// TwinCAT 3 PLC project cryo
// Title: ESO LDC Cryo Library
// Company: ESO
// ProjectVersion: 0.0.0.10
// ProgramVersion: 3.1.4022.4
// libraries:
//   ESO LDC Comm Tcp Library, * (ESO)
//   Tc2_SerialCom, * (Beckhoff Automation GmbH)
//   Tc2_Standard, * (Beckhoff Automation GmbH)
//   Tc2_System, * (Beckhoff Automation GmbH)
//   Tc2_Utilities, * (Beckhoff Automation GmbH)
//   Tc3_Module, * (Beckhoff Automation GmbH)
//   VisuDialogs, * (System)
//   ESO LDC Comm Common Library,0.2.0.2,ESO
//   ESO LDC Comm Serial Library,0.2.0.2,ESO
//   VisuSymbols,3.5.10.0,System
// project tree:
//   / ClassDiagram.TcCD (not stored), ClassDiagram_All.TcCD (not stored), ClassDiagram_Sensors.TcCD (not stored), GlobalTextList.TcGTLO, ImagePool.TcIPO (not stored), PlcTask.TcTTO, Visualization Manager.TcVMO (not stored)
//   DUTs/Enumerations/Actuators/ E_CRYO_BIN_ACT_CMD.TcDUT, E_CRYO_BIN_ACT_FEEDBACK.TcDUT, E_CRYO_BIN_ACT_FEEDBACK_STATE.TcDUT, E_CRYO_BIN_ACT_STATE.TcDUT, E_CRYO_BIN_CTRL_ACTION.TcDUT, E_CRYO_BIN_CTRL_STATE.TcDUT, E_CRYO_CTRL_CMD.TcDUT, E_CRYO_CTRL_STATE.TcDUT, E_CRYO_GEN_CTRL_EVENT.TcDUT
//   DUTs/Enumerations/Coolers/ E_CRYO_CPA_ALARM.TcDUT, E_CRYO_CPA_CMDS.TcDUT, E_CRYO_CPA_DIAG_IDX.TcDUT, E_CRYO_CRYOTELGT_CMD.TcDUT, E_CRYO_CRYOTELGT_STATE.TcDUT
//   DUTs/Enumerations/Misc/ E_CRYO_ALARM_IDX.TcDUT, E_CRYO_ALARM_LEVEL.TcDUT, E_CRYO_THLD_MODE.TcDUT, E_CRYO_VOTE.TcDUT
//   DUTs/Enumerations/Pumps/ E_CRYO_PUMP_STATE.TcDUT, E_ECODRY_VERSION.TcDUT
//   DUTs/Enumerations/Sensors/ E_CRYO_SBG232_SENSOR_TYPE.TcDUT, E_CRYO_SENSOR_TYPE_PRESS.TcDUT, E_CRYO_SENSOR_TYPE_TEMP.TcDUT, E_CRYO_SIM_SENS_CMD.TcDUT
//   DUTs/Enumerations/Subsystems/Evacuation/ E_CRYO_EVAC_PRESSURES_50000.TcDUT, E_CRYO_EVAC_STATE.TcDUT, E_CRYO_EVAC_STATE_50000.TcDUT, E_CRYO_EVAC_SYS_STATE.TcDUT, E_CRYO_EVAC_VALVES_50000.TcDUT
//   DUTs/Structures/Actuators/ T_CRYO_BIN_ACT_STATUS.TcDUT, T_CRYO_BIN_CTRL_STATUS.TcDUT, T_CRYO_GEN_CTRL_STATUS_BASE.TcDUT
//   DUTs/Structures/Coolers/ T_CRYO_CPA_ACTIVE_LIMITS.TcDUT, T_CRYO_CPA_CFG.TcDUT, T_CRYO_CPA_CTRL.TcDUT, T_CRYO_CPA_DIAG_CFG.TcDUT, T_CRYO_CPA_INFO.TcDUT, T_CRYO_CPA_STAT.TcDUT, T_CRYO_CRYOTELGT_CFG.TcDUT, T_CRYO_CRYOTELGT_CMD.TcDUT, T_CRYO_CRYOTELGT_CTRL.TcDUT, T_CRYO_CRYOTELGT_STAT.TcDUT
//   DUTs/Structures/Misc/ T_CRYO_VOTE_LIST.TcDUT
//   DUTs/Structures/Pumps/ T_CRYO_PUMP_ATM2303M_CFG.TcDUT, T_CRYO_PUMP_ATM2303M_STAT.TcDUT, T_CRYO_PUMP_BASE_CFG.TcDUT, T_CRYO_PUMP_BASE_CTRL.TcDUT, T_CRYO_PUMP_BASE_STAT.TcDUT, T_CRYO_PUMP_CMD.TcDUT, T_CRYO_PUMP_HIPACE30_CFG.TcDUT, T_CRYO_PUMP_HIPACE30_STAT.TcDUT, T_CRYO_PUMP_MODBUS_CFG.TcDUT, T_CRYO_PUMP_MODBUS_CTRL.TcDUT, T_CRYO_PUMP_MODBUS_STAT.TcDUT, T_CRYO_PUMP_MVP030_CFG.TcDUT, T_CRYO_PUMP_MVP030_STAT.TcDUT, T_CRYO_PUMP_SERIAL_CFG.TcDUT
//   DUTs/Structures/Sensors/ T_CRYO_IOLINK_SENSOR_STATUS.TcDUT, T_CRYO_PRESSURE_STATUS.TcDUT, T_CRYO_PRESSURE_VOTE_STATUS.TcDUT, T_CRYO_PT100_OHM2C_REC.TcDUT, T_CRYO_SBG232_STAT.TcDUT, T_CRYO_SENSOR_STATUS.TcDUT, T_CRYO_SENSOR_STATUS_PRESS.TcDUT, T_CRYO_SENSOR_STATUS_TEMP.TcDUT, T_CRYO_TEMPERATURE_STATUS.TcDUT
//   DUTs/Structures/Subsystems/Evacuation/ T_CRYO_EVACUATION_SYSTEM_STATUS.TcDUT, T_CRYO_EVAC_CFG.TcDUT, T_CRYO_EVAC_CFG_50000.TcDUT, T_CRYO_EVAC_CTRL.TcDUT, T_CRYO_EVAC_CTRL_50000.TcDUT, T_CRYO_EVAC_STAT.TcDUT, T_CRYO_EVAC_STAT_50000.TcDUT, T_CRYO_EVAC_SYS_INPUT.TcDUT
//   DUTs/Structures/System/ T_CRYO_CFG.TcDUT, T_CRYO_CTRL.TcDUT, T_CRYO_LOG.TcDUT, T_CRYO_STAT.TcDUT
//   POUs/Actuators/ FB_CRYO_ACTUATOR_CMD.TcPOU, FB_CRYO_CMD_OVERRIDE.TcPOU, FB_CRYO_BIN_ACT.TcPOU, FB_CRYO_BIN_CTRL.TcPOU, FB_CRYO_GEN_CTRL_BASE.TcPOU, FB_CRYO_CCC_CTRL.TcPOU, FB_CRYO_HEATER_CTRL.TcPOU, FB_CRYO_LN2_CTRL.TcPOU, FB_CRYO_VALVE_CTRL.TcPOU
//   POUs/Comm/ FB_MODBUS_COMM_CPA.TcPOU
//   POUs/Coolers/ FB_CRYO_CPA.TcPOU, FB_CRYO_CRYOTELGT.TcPOU, FB_RS_COMM_CRYOTELGT.TcPOU, FB_SIM_RS_COMM_CRYOTELGT.TcPOU
//   POUs/ MAIN.TcPOU
//   POUs/Pumps/ FB_CRYO_PUMP_ATH2303M.TcPOU, FB_CRYO_PUMP_BASE.TcPOU, FB_CRYO_PUMP_ECODRY.TcPOU, FB_CRYO_PUMP_HIPACE30.TcPOU, FB_CRYO_PUMP_MODBUS.TcPOU, FB_CRYO_PUMP_MVP030.TcPOU, FB_CRYO_PUMP_SERIAL.TcPOU
//   POUs/Sensors/ FB_CRYO_PRESSURE.TcPOU, FB_CRYO_PRESSURE_VOTE.TcPOU, FB_CRYO_SBG232.TcPOU, FB_CRYO_SENSOR_BASE.TcPOU, FB_CRYO_SENSOR_PRESSURE.TcPOU, FB_CRYO_SENSOR_TEMPERATURE.TcPOU, FB_CRYO_TEMPERATURE.TcPOU
//   POUs/Simulation/ FB_CRYO_SIM_CTRL.TcPOU, FB_CRYO_SIM_SBG232.TcPOU, FB_CRYO_SIM_TEMPERATURE.TcPOU, FB_CRYO_SIM_PRESSURE.TcPOU, FB_CRYO_SIM_SINE.TcPOU, FB_SIM_MODBUS_COMM_CPA.TcPOU
//   POUs/Subsystems/Evacuation/ FB_CRYO_EVACUATION_SYSTEM.TcPOU, FB_CRYO_EVAC_BASE.TcPOU, FB_CRYO_EVAC_BASE_50000.TcPOU
//   POUs/Subsystems/Examples/Evacuation/ FB_CRYO_EVAC_ECODRY_ATH2303M.TcPOU, FB_CRYO_EVAC_MICADO.TcPOU, FB_CRYO_EVAC_PDS.TcPOU, FB_SIM_MICADO_PUMPS.TcPOU, FB_SIM_MICADO_VALVES.TcPOU
//   POUs/Subsystems/Examples/LN2_Precooling/ FB_CRYO_LN2_PRECOOL.TcPOU, FB_SIM_LN2_PRECOOL.TcPOU
//   POUs/System/ FB_CRYO_CTRL.TcPOU
//   POUs/Utilities/ FB_CRYO_THLD_BASE.TcPOU
//   VISUs/GUIs/ GUI_ATH2303M_EVAC_LAB.TcVIS, GUI_CMD_OVERRIDE.TcVIS, GUI_CPA.TcVIS, GUI_CRYO.TcVIS, GUI_CRYOTELGT.TcVIS, GUI_ECODRY_V01_EVAC_LAB.TcVIS, GUI_EVAC_LAB.TcVIS, GUI_EVAC_MICADO.TcVIS, GUI_EVAC_PDS.TcVIS, GUI_HIPACE_30_EVAC_PDS.TcVIS, GUI_IRATEC.TcVIS, GUI_MICADO_Valves.TcVIS, GUI_MVP030_EVAC_PDS.TcVIS, GUI_P2_OVERRIDE.TcVIS, GUI_Pressures.TcVIS, GUI_PVV1_CMD.TcVIS, GUI_SBG232.TcVIS, GUI_SBG232_SIM.TcVIS, GUI_T2_OVERRIDE.TcVIS
//   VISUs/Templates/ GUI_TEMPLATE_ACTUATOR_CMD.TcVIS, GUI_TEMPLATE_ACTUATOR_ENG.TcVIS, GUI_TEMPLATE_SENSOR_SIM_OVERRIDE.TcVIS, GUI_TEMPLATE_ATH2303M.TcVIS, GUI_TEMPLATE_CMD_OVERRIDE.TcVIS, GUI_TEMPLATE_CRYOTELGT.TcVIS, GUI_TEMPLATE_CRYO_CPA.TcVIS, GUI_TEMPLATE_CRYO_EVAC_BASE.TcVIS, GUI_TEMPLATE_ECODRY_V01.TcVIS, GUI_TEMPLATE_HIPACE_30.TcVIS, GUI_TEMPLATE_MVP030.TcVIS, GUI_TEMPLATE_SBG232.TcVIS, GUI_TEMPLATE_TEMP_OVERRIDE.TcVIS, GUI_TEMPLATE_PRESS_OVERRIDE.TcVIS
// real-time tasks:
//   TASK PlcTask: cycle T#1ms, priority 20, ADS port 350
//   TASK VISU_TASK: cycle T#200000us, priority 30, ADS port 351
// motion (NC):
//   TASK NC-Task 1 SAF: cycle T#2ms, priority 4, ADS port 501
//   TASK NC-Task 1 SVB: cycle T#10ms, priority 8, ADS port 511
// I/O:
//   DEVICE Device 1 (EtherCAT) (disabled), AmsNetId 134.171.34.120.2.1
//     Term 1 (EK1200) [EK1200-5000 EtherCAT Power supply (2A E-Bus)]
//       Term 2 (EL2008) [EL2008 8Ch. Dig. Output 24V, 0.5A]
//       Term 3 (EL3162) [EL3162 2Ch. Ana. Input 0-10V]
//       Term 4 (EL1004) [EL1004 4Ch. Dig. Input 24V, 3ms]
//       Term 5 (EL1004) [EL1004 4Ch. Dig. Input 24V, 3ms]
//       Term 6 (EL2622) [EL2622 2Ch. Relay Output, NO (230V AC / 30V DC)]
//       Term 7 (EL6022) [EL6022 Interface 2Ch. (RS422/485)]
//       Term 8 (EL6002) [EL6002 Interface 2Ch. (RS232)]
//       Term 9 (EL9011) [EL9011 End Terminal]
//   DEVICE Device 5 (EtherCAT) (disabled), AmsNetId 134.171.34.120.6.1
//     Term 10 (EK1100) [EK1100 EtherCAT Coupler (2A E-Bus)]
//       Term 11 (EL6224) [EL6224 (IO Link Master)]
//       Term 12 (EL1808) [EL1808 8Ch. Dig. Input 24V, 3ms]
//       Term 13 (EL1808) [EL1808 8Ch. Dig. Input 24V, 3ms]
//       Term 14 (EL2808) [EL2808 8Ch. Dig. Output 24V, 0.5A]
//       Term 15 (EL2652) [EL2652 2Ch. Relay Output, CO (230V AC / 30V DC)]
//       Term 16 (EL2652) [EL2652 2Ch. Relay Output, CO (230V AC / 30V DC)]
//       Term 17 (EL6022) [EL6022 Interface 2Ch. (RS422/485)]
//       Term 18 (EL6022) [EL6022 Interface 2Ch. (RS422/485)]
//       Term 10 (EL9011) [EL9011 End Terminal]
// variable links:
//   cryo/cryo Instance <-> cryo/cryo Instance
//     PlcTask Inputs/MAIN.evac_micado.GBV.Actuator.i_bOFF <-> PlcTask Outputs/MAIN.mic_valves.q_bOFF_GBV
//     PlcTask Inputs/MAIN.evac_micado.GBV.Actuator.i_bON <-> PlcTask Outputs/MAIN.mic_valves.q_bON_GBV
//     PlcTask Inputs/MAIN.evac_micado.GBV.Actuator.i_nCouplerState <-> PlcTask Outputs/MAIN.q_nCouplerState
//     PlcTask Inputs/MAIN.evac_micado.PVV{1..4}.Actuator.i_bOFF <-> PlcTask Outputs/MAIN.mic_valves.q_bOFF_PVV{1..4}  (4 links)
//     PlcTask Inputs/MAIN.evac_micado.PVV{1..4}.Actuator.i_bON <-> PlcTask Outputs/MAIN.mic_valves.q_bON_PVV{1..4}  (4 links)
//     PlcTask Inputs/MAIN.evac_micado.PVV{1..4}.Actuator.i_nCouplerState <-> PlcTask Outputs/MAIN.q_nCouplerState  (4 links)
//     PlcTask Inputs/MAIN.evac_micado.rp.i_bRunning <-> PlcTask Outputs/MAIN.mic_pumps.q_PVP_Running
//     PlcTask Inputs/MAIN.evac_micado.sensor_VAG1.i_nStatus <-> PlcTask Outputs/MAIN.pSim.q_nStatus
//     PlcTask Inputs/MAIN.evac_micado.sensor_VAG2.i_nStatus <-> PlcTask Outputs/MAIN.pSim.q_nStatus
//     PlcTask Inputs/MAIN.evac_micado.sensor_VAG3.i_nStatus <-> PlcTask Outputs/MAIN.pSim.q_nStatus
//     PlcTask Inputs/MAIN.evac_micado.sensor_VAG1.i_nValue <-> PlcTask Outputs/MAIN.q_nVAG1
//     PlcTask Inputs/MAIN.evac_micado.sensor_VAG2.i_nValue <-> PlcTask Outputs/MAIN.q_nVAG2
//     PlcTask Inputs/MAIN.evac_micado.sensor_VAG3.i_nValue <-> PlcTask Outputs/MAIN.q_nVAG3
//     PlcTask Inputs/MAIN.evac_micado.tp.i_bReady <-> PlcTask Outputs/MAIN.mic_pumps.q_TMP_Ready
//     PlcTask Inputs/MAIN.evac_micado.tp.i_bSpeed100 <-> PlcTask Outputs/MAIN.mic_pumps.q_TMP_Speed100
//     PlcTask Inputs/MAIN.ln2_ctrl.valve.Actuator.i_bON <-> PlcTask Outputs/MAIN.ln2_ctrl.valve.Actuator.q_bCtrl
//     PlcTask Inputs/MAIN.ln2_ctrl.valve.Actuator.i_nCouplerState <-> PlcTask Outputs/MAIN.Cryo_Ctrl.q_nStateDummy
//     PlcTask Inputs/MAIN.mic_valves.i_bON_GBV <-> PlcTask Outputs/MAIN.evac_micado.GBV.Actuator.q_bCtrl
//     PlcTask Inputs/MAIN.mic_valves.i_bON_PVV{1..4} <-> PlcTask Outputs/MAIN.evac_micado.PVV{1..4}.Actuator.q_bCtrl  (4 links)
//     PlcTask Inputs/MAIN.sbg232_sim.i_ArrPortProcessData <-> PlcTask Outputs/MAIN.SIM_sbg232.q_ArrPortProcessData
//     PlcTask Inputs/MAIN.sbg232_sim.i_nCouplerState <-> PlcTask Outputs/MAIN.SIM_sbg232.q_nCouplerState
//     PlcTask Inputs/MAIN.sbg232_sim.i_nDeviceStateInputCh <-> PlcTask Outputs/MAIN.SIM_sbg232.q_nDeviceStateInputCh
//     PlcTask Inputs/MAIN.sensor_VAGF1.i_nStatus <-> PlcTask Outputs/MAIN.pSim.q_nStatus
//     PlcTask Inputs/MAIN.sensor_VAGF2.i_nStatus <-> PlcTask Outputs/MAIN.pSim.q_nStatus
//     PlcTask Inputs/MAIN.sensor_VAGF1.i_nValue <-> PlcTask Outputs/MAIN.q_nVAGF1
//     PlcTask Inputs/MAIN.sensor_VAGF2.i_nValue <-> PlcTask Outputs/MAIN.q_nVAGF2
//     PlcTask Inputs/MAIN.sensor_VAGG1.i_nStatus <-> PlcTask Outputs/MAIN.pSim.q_nStatus
//     PlcTask Inputs/MAIN.sensor_VAGG2.i_nStatus <-> PlcTask Outputs/MAIN.pSim.q_nStatus
//     PlcTask Inputs/MAIN.sensor_VAGG1.i_nValue <-> PlcTask Outputs/MAIN.q_nVAGG1
//     PlcTask Inputs/MAIN.sensor_VAGG2.i_nValue <-> PlcTask Outputs/MAIN.q_nVAGG2

CONFIGURATION cryo
    RESOURCE PLC ON TwinCAT3
        TASK PlcTask(INTERVAL := T#1ms, PRIORITY := 20);
        PROGRAM MAIN WITH PlcTask : MAIN;
    END_RESOURCE
END_CONFIGURATION

// ---- DUTs/Enumerations/Actuators/E_CRYO_BIN_ACT_CMD.TcDUT
{attribute 'qualified_only'}
{attribute 'strict'}
TYPE E_CRYO_BIN_ACT_CMD :
(
	NONE	:= 0,
	OFF 	:= 1,
	ON		:= 2
);
END_TYPE

// ---- DUTs/Enumerations/Actuators/E_CRYO_BIN_ACT_FEEDBACK.TcDUT
{attribute 'qualified_only'}
{attribute 'strict'}
TYPE E_CRYO_BIN_ACT_FEEDBACK :
(
	ON_AND_OFF	:= 0,	// There are two separate signals: ON (i_bON) and OFF (i_bOFF)
	ON_ONLY 	:= 1	// Feedback exists only for ON signal
);
END_TYPE

// ---- DUTs/Enumerations/Actuators/E_CRYO_BIN_ACT_FEEDBACK_STATE.TcDUT
{attribute 'qualified_only'}
{attribute 'strict'}
TYPE E_CRYO_BIN_ACT_FEEDBACK_STATE :
(
	OFF		:= 0,
	ON	 	:= 1,
	ERROR	:= 2
);
END_TYPE

// ---- DUTs/Enumerations/Actuators/E_CRYO_BIN_ACT_STATE.TcDUT
{attribute 'qualified_only'}
{attribute 'strict'}
TYPE E_CRYO_BIN_ACT_STATE :
(
	NONE := 0,
	OFF,
	SWITCHING_ON,
	ON,
	SWITCHING_OFF,
	ERROR
);
END_TYPE

// ---- DUTs/Enumerations/Actuators/E_CRYO_BIN_CTRL_ACTION.TcDUT
TYPE E_CRYO_BIN_CTRL_ACTION :
(
	NONE := 0,
	OFF,
	ON
);
END_TYPE

// ---- DUTs/Enumerations/Actuators/E_CRYO_BIN_CTRL_STATE.TcDUT
{attribute 'qualified_only'}
{attribute 'strict'}
TYPE E_CRYO_BIN_CTRL_STATE :
(
	NONE := 0,
	OFF,					// Controller OFF, Actuator OFF
	ACTIVE_SWITCHING_ON,	// Activating Controller
	ACTIVE_OFF,				// Controller active, Actuator OFF
	ACTIVE_ON,				// Controller active, Actuator ON
	ACTIVE_SWITCHING_OFF,	// Switching Actuator OFF and going OFF with Controller
	ERROR					// Actuator failure
);
END_TYPE

// ---- DUTs/Enumerations/Actuators/E_CRYO_CTRL_CMD.TcDUT
{attribute 'qualified_only'}
{attribute 'strict'}
TYPE E_CRYO_CTRL_CMD :
(
	NONE	:= 0,
	PRECOOL,
	COOL,
	WARM_UP,
	REPRESSURIZE
);
END_TYPE

// ---- DUTs/Enumerations/Actuators/E_CRYO_CTRL_STATE.TcDUT
{attribute 'qualified_only'}
{attribute 'strict'}
TYPE E_CRYO_CTRL_STATE :
(
	NONE 			:= 0,
	WARM_PRESS,				// Warm & Pressurized
	WARM_VACUUM,			// Warm & Vacuum
	PRE_COOLING,			// Pre_cooling
	PRE_COOLED,				// Pre_cooled
	COOLING_DOWN,			// Cooling down
	COLD,					// Cold, i.e. fully operational
	WARMING_UP,				// Warming up
	REPRESSURIZING,			// Re-pressurizing			
	ERROR					// Controller failure
);
END_TYPE

// ---- DUTs/Enumerations/Actuators/E_CRYO_GEN_CTRL_EVENT.TcDUT
{attribute 'qualified_only'}
{attribute 'strict'}
TYPE E_CRYO_GEN_CTRL_EVENT :
(
	NONE := 0,
	ENABLE,
	DISABLE,
	OFF,
	IS_OFF,
	ON,
	IS_ON,
	ERROR
);
END_TYPE

// ---- DUTs/Enumerations/Coolers/E_CRYO_CPA_ALARM.TcDUT
{attribute 'qualified_only'}
{attribute 'strict'}
TYPE E_CRYO_CPA_ALARM :
(
	NONE := 0,
	LOW,
	HIGH
);
END_TYPE

// ---- DUTs/Enumerations/Coolers/E_CRYO_CPA_CMDS.TcDUT
{attribute 'qualified_only'}
{attribute 'strict'}
TYPE E_CRYO_CPA_CMDS :
(
	NONE	:= 0,
	START	:= 21,
	STOP
);
END_TYPE

// ---- DUTs/Enumerations/Coolers/E_CRYO_CPA_DIAG_IDX.TcDUT
{attribute 'qualified_only'}
{attribute 'strict'}
TYPE E_CRYO_CPA_DIAG_IDX :
(
	WATER_IN	:= 0,
	WATER_OUT,
	OIL_TEMP,
	HELIUM_TEMP,
	HELIUM_LOW_PRESS_OP,
	HELIUM_HIGH_PRESS_OP,
	HELIUM_DELTA_PRESS,
	HELIUM_STATIC_LOW_PRESS,
	HELIUM_STATIC_HIGH_PRESS
);
END_TYPE

// ---- DUTs/Enumerations/Coolers/E_CRYO_CRYOTELGT_CMD.TcDUT
{attribute 'qualified_only'}
{attribute 'strict'}
TYPE E_CRYO_CRYOTELGT_CMD :
(
	NONE := 0,
	OFF,
	ON,
	SET_POWER
);
END_TYPE

// ---- DUTs/Enumerations/Coolers/E_CRYO_CRYOTELGT_STATE.TcDUT
{attribute 'qualified_only'}
{attribute 'strict'}
TYPE E_CRYO_CRYOTELGT_STATE :
(
	OFF := 0,
	STARTING,
	ON,
	STOPPING,
	ERROR
);
END_TYPE

// ---- DUTs/Enumerations/Misc/E_CRYO_ALARM_IDX.TcDUT
{attribute 'qualified_only'}
{attribute 'strict'}
TYPE E_CRYO_ALARM_IDX :
(
	ALARM_LOW 		:= 1,
	WARNING_LOW		:= 2,
	WARNING_HIGH	:= 3,
	ALARM_HIGH		:= 4
);
END_TYPE

// ---- DUTs/Enumerations/Misc/E_CRYO_ALARM_LEVEL.TcDUT
{attribute 'qualified_only'}
{attribute 'strict'}
TYPE E_CRYO_ALARM_LEVEL :
(
	ALARM_LOW 		:= -2,
	WARNING_LOW		:= -1,
	NORMAL			:= 0,
	WARNING_HIGH	:= 1,
	ALARM_HIGH		:= 2
);
END_TYPE

// ---- DUTs/Enumerations/Misc/E_CRYO_THLD_MODE.TcDUT
{attribute 'qualified_only'}
{attribute 'strict'}
TYPE E_CRYO_THLD_MODE :
(
	FIXED := 0,		// Thresholds as set with input parameters
	ACTIVE,			// Thresholds are calculated based on input parameter(s)
	LAST_ACTIVE		// Thresholds are kept at last ACTIVE levels 
);
END_TYPE

// ---- DUTs/Enumerations/Misc/E_CRYO_VOTE.TcDUT
{attribute 'qualified_only'}
{attribute 'strict'}
TYPE E_CRYO_VOTE :
(
	V_AVE	:= 0,
	V_MIN,
	V_MAX,
	V_1oo2,
	V_2oo3,
	V_3oo5
);
END_TYPE

// ---- DUTs/Enumerations/Pumps/E_CRYO_PUMP_STATE.TcDUT
{attribute 'qualified_only'}
{attribute 'strict'}
TYPE E_CRYO_PUMP_STATE :
(
	OFF := 0,
	STARTING,
	ON,
	STOPPING,
	ERROR
);
END_TYPE

// ---- DUTs/Enumerations/Pumps/E_ECODRY_VERSION.TcDUT
{attribute 'qualified_only'}
{attribute 'strict'}
TYPE E_ECODRY_VERSION :
(
	V01 := 0,
	V21_22
);
END_TYPE

// ---- DUTs/Enumerations/Sensors/E_CRYO_SBG232_SENSOR_TYPE.TcDUT
{attribute 'qualified_only'}
{attribute 'strict'}
TYPE E_CRYO_SBG232_SENSOR_TYPE :
(
	NONE := 0,
	FLOW,
	TEMP
);
END_TYPE

// ---- DUTs/Enumerations/Sensors/E_CRYO_SENSOR_TYPE_PRESS.TcDUT
{attribute 'qualified_only'}
{attribute 'strict'}
TYPE E_CRYO_SENSOR_TYPE_PRESS :
(
	NONE 		:= 0,
	PKR_250		:= 1,	// Pfeiffer PKR250 & PKR251 have the same formula
	CMR_361		:= 2,	// Pfeiffer CMR361
	WRG_D_NW25	:= 3,	// Edwards WRG-D-NW25
	PKR_360		:= 4	// Pfeiffer PKR360
);
END_TYPE

// ---- DUTs/Enumerations/Sensors/E_CRYO_SENSOR_TYPE_TEMP.TcDUT
{attribute 'qualified_only'}
{attribute 'strict'}
TYPE E_CRYO_SENSOR_TYPE_TEMP :
(
	NONE 	:= 0,
	PT100	:= 1
);
END_TYPE

// ---- DUTs/Enumerations/Sensors/E_CRYO_SIM_SENS_CMD.TcDUT
{attribute 'qualified_only'}
{attribute 'strict'}
TYPE E_CRYO_SIM_SENS_CMD :
(
	NONE	:= 0,
	SET 	:= 1,	// Set value
	RAMP	:= 2,	// Ramp value
	SINE	:= 3	// Vary value as SINE signal
);
END_TYPE

// ---- DUTs/Enumerations/Subsystems/Evacuation/E_CRYO_EVAC_PRESSURES_50000.TcDUT
{attribute 'qualified_only'}
{attribute 'strict'}
TYPE E_CRYO_EVAC_PRESSURES_50000 :
(
	NONE := 0,
	VAG1,		
	VAG2,		
	VAG3,		
	VAGF,		
	VAGG		
);
END_TYPE

// ---- DUTs/Enumerations/Subsystems/Evacuation/E_CRYO_EVAC_STATE.TcDUT
{attribute 'qualified_only'}
{attribute 'strict'}
TYPE E_CRYO_EVAC_STATE :
(
	NONE := 0,				// Undefined state.
	OFF,					// Everything is OFF.
	START_R_PUMP,			// Starting Roughing Pump.
	WAIT_PREVAC,			// Waiting for the prevaccum pressure to be reached.
	OPEN_INSULATION_VALVE,	// Opening Insulation Valve.
	START_T_PUMP,			// Starting Turbo-Molecular Pump.
	WAIT_CRYO_VAC,			// Waiting for the cryo pressure to drop below threshold.
	EVACUATING,				// System is running. Evacuation in progress.
	CLOSE_INSULATION_VALVE,	// Closing Insulation Valve.
	DELAY_STOPPING,			// Delay after closing Insulation valve before stopping pumps.
	STOP_T_PUMP,			// Stopping Turbo-Molecular Pump.
	STOP_R_PUMP,			// Stopping Roughing Pump.
	WAIT_T_PUMP_STOP		// Waiting for the Turbo-Molecular Pump to stop.
);
END_TYPE

// ---- DUTs/Enumerations/Subsystems/Evacuation/E_CRYO_EVAC_STATE_50000.TcDUT
{attribute 'qualified_only'}
{attribute 'strict'}
TYPE E_CRYO_EVAC_STATE_50000 :
(
	NONE := 0,				// Undefined state.
	OFF,					// Everything is OFF.
	START_PVP,				// Starting PreVacuum Pump (Roughing Pump).
	OPEN_GBV,				// Opening gas-ballast valve
	WAIT_VAG3,				// Waiting for VAG3 pressure < 0.1 mbar.
	OPEN_PVV1,				// Opening PVV1 Pre-vacuum Valve.
	WAIT_VAG_1_3,			// Waiting for VAG1 & VAG3 pressure < 0.1 mbar.
	OPEN_PVV2,				// Opening PVV2 Pre-vacuum Valve.
	WAIT_VAG_F_G_1,			// Waiting for VAGF & VAGG pressure < 0.9x0.1 mbar.
	CLOSE_PVV2,				// Closing PVV2 Pre-vacuum Valve.
	CLOSE_PVV1,				// Closing PVV1 Pre-vacuum Valve.
	START_TMP,				// Starting Turbo-Molecular Pump (TMP).
	OPEN_PVV3,				// Opening PVV3 Pre-vacuum Valve.
	WAIT_VAG_2_3,			// Waiting for VAG2 & VAG3 pressure < 0.1 mbar.
	OPEN_PVV4,				// Opening PVV4 Pre-vacuum Valve.
	WAIT_VAG_F_G_2,			// Waiting for VAGF & VAGG pressure < 0.0001 mbar.
	CLOSE_GBV,				// Closing gas-ballast valve
	EVACUATING,				// System is running. Evacuation in progress.
	CLOSE_ALL_VALVES,		// Closing All Valves.
	DELAY_STOPPING,			// Delay after closing valves before stopping pumps.
	STOP_TMP_1,				// Stopping Turbo-Molecular Pump (TMP) - case 1.
	STOP_TMP_2,				// Stopping Turbo-Molecular Pump (TMP) - case 2.
	STOP_PVP,				// Stopping PreVacuum Pump (Roughing Pump).
	WAIT_TMP_STANDSTILL		// Waiting for the Turbo-Molecular Pump to standstill.
);
END_TYPE

// ---- DUTs/Enumerations/Subsystems/Evacuation/E_CRYO_EVAC_SYS_STATE.TcDUT
{attribute 'qualified_only'}
{attribute 'strict'}
TYPE E_CRYO_EVAC_SYS_STATE :
(
	NONE := 0,
	OFF,					// Controller OFF, Valve closed
//	ACTIVE_STARTING_PUMPS,	// Controller ON,  Starting pumps
//	ACTIVE_PUMPS_RUNNING,	// Controller ON,  Pumps running
	ACTIVE_OPENING,			// Controller ON,  Valve opening
	ACTIVE_OPEN,			// Controller ON,  Valve open
	ACTIVE_CLOSING,			// Controller ON,  Valve closing
	ACTIVE_CLOSED,			// Controller ON,  Valve closed
//	ACTIVE_STOPPING_PUMPS,	// Controller ON,  Stopping pumps
	EMERGENCY,				// Controller ON,  Closing valve for safety reason
	ERROR					// Error in the system
);
END_TYPE

// ---- DUTs/Enumerations/Subsystems/Evacuation/E_CRYO_EVAC_VALVES_50000.TcDUT
{attribute 'qualified_only'}
{attribute 'strict'}
TYPE E_CRYO_EVAC_VALVES_50000 :
(
	NONE := 0,
	PVV1,		
	PVV2,		
	PVV3,		
	PVV4,		
	GBV		
);
END_TYPE

// ---- DUTs/Structures/Actuators/T_CRYO_BIN_ACT_STATUS.TcDUT
TYPE T_CRYO_BIN_ACT_STATUS :
STRUCT
	bDone:		BOOL;			// Flag if switch is OK
	bBusy:		BOOL;			// Flag if switch is BUSY
	bError:		BOOL;			// Flag if switch is OK
	bON:		BOOL;			// Flag if switch state is ON
	bOFF:		BOOL;			// Flag if switch state is OFF

	nLastCommand:	E_CRYO_BIN_ACT_CMD		:= E_CRYO_BIN_ACT_CMD.NONE;	// Command
	nState:			E_CRYO_BIN_ACT_STATE	:= E_CRYO_BIN_ACT_STATE.NONE;
	
	sState:		STRING(64);			// State as text
END_STRUCT
END_TYPE

// ---- DUTs/Structures/Actuators/T_CRYO_BIN_CTRL_STATUS.TcDUT
TYPE T_CRYO_BIN_CTRL_STATUS :
STRUCT
	bDone:		BOOL;			// Flag if controller is OK
	bBusy:		BOOL;			// Flag if controller is BUSY
	bError:		BOOL;			// Flag if controller is OK
	bActive:	BOOL;			// Flag if controller is ACTIVE
	bActON:		BOOL;			// Flag if actuator is ON
	bActOFF:	BOOL;			// Flag if actuator is OFF

	// Generic controller OK flag.
	// Used for problems other than from the actuator.
	// This flag is used for problems coming from controllers
	// that extend the functionality of FB_CRYO_BIN_CTRL.
	bCtrlOK:	BOOL := TRUE;		

	nCycleCounter:	UDINT := 0;
	nState:			E_CRYO_BIN_CTRL_STATE	:= E_CRYO_BIN_CTRL_STATE.NONE;

	sState:		STRING(64);		// State as text
END_STRUCT
END_TYPE

// ---- DUTs/Structures/Actuators/T_CRYO_GEN_CTRL_STATUS_BASE.TcDUT
TYPE T_CRYO_GEN_CTRL_STATUS_BASE :
STRUCT
	bDone:			BOOL;			// Flag if controller is OK
	bBusy:			BOOL;			// Flag if controller is BUSY
	bError:			BOOL;			// Flag if controller is in ERROR state
	bActive:		BOOL;			// Flag if controller is ACTIVE

	nCycleCounter:	UDINT := 0;
	nState:			E_CRYO_BIN_CTRL_STATE	:= E_CRYO_BIN_CTRL_STATE.NONE;

	sState:			STRING(64);		// State as text
	sError:			STRING(64);		// Error as text
END_STRUCT
END_TYPE

// ---- DUTs/Structures/Coolers/T_CRYO_CPA_ACTIVE_LIMITS.TcDUT
TYPE T_CRYO_CPA_ACTIVE_LIMITS :
STRUCT
	rErrorLow:		REAL;	// Error for Low  range
	rAlarmLow:		REAL;	// Alarm for Low  range MAX(CRYOMECH,ESO)
	rAlarmHigh:		REAL;	// Alarm for High range MIN(CRYOMECH,ESO)
	rErrorHigh:		REAL;	// Error for High range
END_STRUCT
END_TYPE

// ---- DUTs/Structures/Coolers/T_CRYO_CPA_CFG.TcDUT
TYPE T_CRYO_CPA_CFG EXTENDS T_RS_BASE_CFG:
STRUCT
	// Register Addresses
	nAddrCommon:		INT	:= 16#0001;	// 16#0001

	// Number of bytes to read
	// These are ONLY data bytes. Total bytes to read is higher (+5) 
	nWordsCommon:		INT	:= 32;	// 64w=128 bytes
	
	nSlaveID:			BYTE := 1;	// Slave ID
	bDevUsed:			BOOL := TRUE;	

	nPosOffset:	INT	:= 0;	// byte position in the buffer - for testing
	
	// Thresholds for 'service due' warnings.
	// Warning 'Service due in xxx hours' will appear if less than the threshold is left.
	lrServiceDue_Compressor:	LREAL	:= 1000.0; // hours
	lrServiceDue_PulseTube:		LREAL	:= 2000.0; // hours
	
	
//
// Alarms and warnings
//
	
(*
7.7.7 Error and warning set points
==================================
"High pressure too High!" YES 400 PSIG (27.6bar) 375 PSIG (25.9 bar)
"High pressure too Low!" YES 150 PSIG (10.3bar) 170 PSIG (11.7 bar)
“Low Pressure Too Low!” YES 40 PSIG (2.8 bar) 50 PSIG (3.4 bar)
“Low Pressure Too High!" YES 250 PSIG (17.2 bar) 240 PSIG (16.5 bar)
"Delta Pressure Too High!" YES 400 PSIG (27.6bar) 275 PSIG (19 bar)
"Delta Pressure Too Low!" YES 50 PSIG (3.4 bar) 75 PSIG (5.2 bar)
"Static Pressure Too High!" YES 300 PSIG (20.7 bar) 280 PSIG (19.3 bar)
"Static Pressure Too Low!" YES 100 PSIG (6.9 bar) 170 PSIG (11.7 bar)
"Water In Temp Too High" YES 110°F (43°C) 80°F (27°C)
"Water In Temp Too Low" YES 40°F (4°C) 50°F (10°C)
“Water Out Temp Too High!” YES 125°F (52°C) 110°F (43°C)
"Water Out Temp Too Low" YES 40°F (4°C) 50°F (10°C)
“Helium Temp Too High!” YES 190°F (88°C) 120°F (49°C)
“Helium Temp Too Low!" YES 40°F (4°C) 50°F (10°C)
“Oil Temp Too High!” YES 125°F (52°C) 110°F (43°C)
“Oil Temp Too Low!" YES 40°F (4°C) 50°F (10°C)
“Compressor Motor Current Too Low!” YES < 5A ≥ 5 A


Warning Description Trip / Clear
================================
"High Pressure Running High!" 375 PSIG (25.9bar)
"High Pressure Running Low!" 170 PSIG (11.7bar)
“Low Pressure Running Low!” 50 PSIG (3.4 bar)
“Low Pressure Running High!" 240 PSIG (16.5 bar)
"Delta Pressure Running High!" 275 PSIG (19.0bar)
"Delta Pressure Running Low!" 75 PSIG (5.2 bar)
"Static Pressure Running High!" 280 PSIG (19.3 bar)
"Static Pressure Running Low!" 170 PSIG (11.7 bar)
"Water In Temp Running High" 85°F (29°C)
"Water In Temp Running Low" 45°F (7°C)
“Water Out Temp Running High!” 110°F (43°C)
"Water Out Temp Running Low" 45°F (7°C)
“Helium Temp Running High!” 170°F (77°C)
“Helium Temp Running Low!" 45°F (7°C)
“Oil Temp Running High!” 110°F (43°C)
“Oil Temp Running Low!" 45°F (7°C)

*)
	//
	// Diagnostics configuration.
	// Low and high limits for alarms and errors.
	//
	aDiag:	ARRAY [0..8] OF T_CRYO_CPA_DIAG_CFG := [ 
		(sLabel:='Water IN',	sUnits:='ºC',	nBitLow:=1, nBitHigh:=0,
			rErrorLow:=4.0, 		rAlarmLow_CPA:=7.0,	rAlarmLow_ESO:=7.0,	
			rAlarmHigh_ESO:=27.0,	rAlarmHigh_CPA:=29.0,	rErrorHigh:=43.0),
		(sLabel:='Water OUT',	sUnits:='ºC', 	nBitLow:=3, nBitHigh:=2,
			rErrorLow:=4.0, 		rAlarmLow_CPA:=7.0, 	rAlarmLow_ESO:=7.0, 
			rAlarmHigh_ESO:=50.0, 	rAlarmHigh_CPA:=43.0, 	rErrorHigh:=52.0),
		(sLabel:='Oil temperature', sUnits:='ºC',  	nBitLow:=5, nBitHigh:=4,
			rErrorLow:=4.0, 		rAlarmLow_CPA:=7.0, 	rAlarmLow_ESO:=7.0, 
			rAlarmHigh_ESO:=50.0, 	rAlarmHigh_CPA:=43.0, 	rErrorHigh:=52.0),
		(sLabel:='Helium temperature', 				sUnits:='ºC',  	nBitLow:=7, nBitHigh:=6,
			rErrorLow:=4.0, 		rAlarmLow_CPA:=7.0, 	rAlarmLow_ESO:=7.0, 
			rAlarmHigh_ESO:=80.0, 	rAlarmHigh_CPA:=77.0, 	rErrorHigh:=88.0),
		(sLabel:='Operational Helium low pressure',	sUnits:='bar',  	nBitLow:=9, nBitHigh:=8,
			rErrorLow:=2.8, 		rAlarmLow_CPA:=3.4, 	rAlarmLow_ESO:=4.0, 
			rAlarmHigh_ESO:=13.0, 	rAlarmHigh_CPA:=16.5, 	rErrorHigh:=17.2),
		(sLabel:='Operational Helium high pressure',	sUnits:='bar',  	nBitLow:=11, nBitHigh:=10,
			rErrorLow:=10.3, 		rAlarmLow_CPA:=11.7, 	rAlarmLow_ESO:=17.0, 
			rAlarmHigh_ESO:=25.0, 	rAlarmHigh_CPA:=25.9, 	rErrorHigh:=27.6),
		(sLabel:='Delta operational Helium pressure',	sUnits:='bar',  	nBitLow:=13, nBitHigh:=12,
			rErrorLow:=3.4, 		rAlarmLow_CPA:=5.2, 	rAlarmLow_ESO:=6.0, 
			rAlarmHigh_ESO:=18.0, 	rAlarmHigh_CPA:=19.0, 	rErrorHigh:=27.6),
		(sLabel:='Static Helium low pressure',			sUnits:='bar',  	nBitLow:=18, nBitHigh:=17,
			rErrorLow:=6.9, 		rAlarmLow_CPA:=11.7, 	rAlarmLow_ESO:=12.0, 
			rAlarmHigh_ESO:=19.0, 	rAlarmHigh_CPA:=19.3, 	rErrorHigh:=20.7),
		(sLabel:='Static Helium high pressure',		sUnits:='bar',  	nBitLow:=18, nBitHigh:=17,
			rErrorLow:=6.9, 		rAlarmLow_CPA:=11.7, 	rAlarmLow_ESO:=12.0, 
			rAlarmHigh_ESO:=19.0, 	rAlarmHigh_CPA:=19.3, 	rErrorHigh:=20.7)];
	
	// Dynamic pressure limits.
	// Limits depend on compressor state 
	// ON 	- Operational pressure
	// OFF - Static pressure
//	stActPressLimit_Low:	T_CRYO_CPA_ACTIVE_LIMITS;
//	stActPressLimit_High:	T_CRYO_CPA_ACTIVE_LIMITS;
	// Array of limits. Dynamically set
	aLimits:	ARRAY [0..6] OF T_CRYO_CPA_ACTIVE_LIMITS;	
	aLimits_OP:	ARRAY [0..6] OF T_CRYO_CPA_ACTIVE_LIMITS;	
	aLimits_ST:	ARRAY [0..6] OF T_CRYO_CPA_ACTIVE_LIMITS;	

	

END_STRUCT
END_TYPE

// ---- DUTs/Structures/Coolers/T_CRYO_CPA_CTRL.TcDUT
TYPE T_CRYO_CPA_CTRL EXTENDS T_RS_BASE_CTRL:
STRUCT
	nDevCommand:	E_CRYO_CPA_CMDS := E_CRYO_CPA_CMDS.NONE;	// CPA specific commands
	bCtrlPulseActive:	BOOL	:= FALSE;	// Switching compressor on/off active

	nSlaveID:	BYTE 	:= 1;						// Modbus Slave ID, 1..247
	nCmdType:	DINT	:= E_MODBUS_CMD_TYPE.READ;	// Command type; 0-Read, 1-Write
	nRegister:	DINT;								// Command register
	nWords:		DINT	:= 1;						// Number of words
	nValue:		DINT;								// Parameter value
	
	
END_STRUCT
END_TYPE

// ---- DUTs/Structures/Coolers/T_CRYO_CPA_DIAG_CFG.TcDUT
TYPE T_CRYO_CPA_DIAG_CFG :
STRUCT
	sLabel:				STRING(56)	:= '';	// Label for Inputs, e.g. 'Water IN'
	sUnits:				STRING(8)	:= '';	// User units
	nBitLow:			INT;	// Bit position in warnings/errors for Low
	nBitHigh:			INT;	// Bit position in warnings/errors for High
	rErrorLow:			REAL;	// Error for Low  range
	rAlarmLow_CPA:		REAL;	// Alarm for Low  range as defined by CRYOMECH
	rAlarmLow_ESO:		REAL;	// Alarm for Low  range as defined by ESO
	rAlarmHigh_ESO:		REAL;	// Alarm for High range as defined by ESO
	rAlarmHigh_CPA:		REAL;	// Alarm for High range as defined by CRYOMECH
	rErrorHigh:			REAL;	// Error for High range
END_STRUCT
END_TYPE

// ---- DUTs/Structures/Coolers/T_CRYO_CPA_INFO.TcDUT
TYPE T_CRYO_CPA_INFO :
STRUCT
(*
	Driver Information

	Change LOG:
*)
	sDate:			STRING(16)	:= '2020-07-14';
	sDescription:	STRING(32) 	:= 'CPA controller';
	sName:			STRING(16)	:= 'FB_CRYO_CPA';
	sPlatform:		STRING(16)	:= 'CoDeSys';
	sSynopsis:		STRING(48)	:= 'EtherCAT PLC CPA controller';
	nVersionMajor:	DINT		:= 1;
	nVersionMinor:	DINT		:= 0;

END_STRUCT
END_TYPE

// ---- DUTs/Structures/Coolers/T_CRYO_CPA_STAT.TcDUT
TYPE T_CRYO_CPA_STAT EXTENDS T_RS_BASE_STAT:
STRUCT
	bSystemOn:				BOOL := FALSE;

	nRetries:				INT := 0;	// Total number of retries in case of communication problems
	
	nInputBuffer: 			ARRAY [0..300] OF BYTE;	// Binary data read from JUMO
	
	// Parameters read from the compressor
	nOperatingState:		INT	:= 0;
	nCompressorRunning:		INT	:= 0;
	lrWarningState:			LREAL	:= 0.0;
	lrAlarmState:			LREAL	:= 0.0;
	lrCoolantInTemp:		LREAL	:= 0.0;
	lrCoolantOutTemp:		LREAL	:= 0.0;
	lrOilTemp:				LREAL	:= 0.0;
	lrHeliumTemp:			LREAL	:= 0.0;
	lrLowPressure:			LREAL	:= 0.0;
	lrLowPressureAverage:	LREAL	:= 0.0;
	lrHighPressure:			LREAL	:= 0.0;
	lrHighPressureAverage:	LREAL	:= 0.0;
	lrDeltaPressureAverage:	LREAL	:= 0.0;
	lrMotorCurrent:			LREAL	:= 0.0;
	lrHoursOfOperation:		LREAL	:= 0.0;
	nPressureScale:			INT		:= 0;
	nTempScale:				INT		:= 0;
	nPanelSerialNumber:		UINT	:= 0;
	nModelMajorMinor:		INT		:= 0;

	// Calculated values
	sOperatingState:		STRING(32);
	sModelNumber:			STRING	:= 'CRYOMECH CPAxxxx';

	sServiceDue_Compressor:	STRING	:= ''; 		// Warning string for compressor service
	sServiceDue_PulseTube:	STRING	:= ''; 		// Warning string for pulse tube service
	

	bServiceDue_Compressor:	BOOL	:= FALSE;	// Warning for compressor service
	bServiceDue_PulseTube:	BOOL	:= FALSE;	// Warning for pulse tube service
	
	wColour_Compressor:		DWORD;	// Warning colour for compressor service
	wColour_PulseTube:		DWORD;	// Warning colour for pulse tube service

	
	
(*	
Input Register 30005: (Errors)
0: No Errors
-1: CoolantInHigh
-2: CoolantInLow
-4: CoolantOutHigh
-8: CoolantOutLow
-16: OilHigh
-32: OilLow
-64: HeliumHigh
-128: HeliumLow
-256: LowPressureHigh
-512: LowPressureLow
-1024: HighPressureHigh
-2048: HighPressureLow
-4096: DeltaPressureHigh
-8192: DeltaPressureLow
-16384: MotorCurrentLow
-32768: ThreePhaseError
-65536: PowerSupplyError
-131072: StaticPressureHigh
-262144: StaticPressureLow
*)
	
	
	// Readings in array
	aReadings:	ARRAY [0..6] OF LREAL;	// For index, see E_CRYO_CPA_DIAG_IDX
	
	// Alarms in array
	arrAlarms:		ARRAY [0..8] OF INT;
	// Errors in array
	arrErrors:		ARRAY [0..8] OF INT;
	
	// Alarm text, e.g. 
	// ‘Alarm: high pressure running high, compressor will shut off at 27.6 bar’
	sAlarm:		STRING(128)	:= '';	
	// Error text, e.g. 
	// ‘Error: high pressure running high, compressor shut off at 27.6 bar’
	sError:		STRING(128)	:= '';	
	sStatusOK:	STRING(128)	:= 'Running Normally';	
	
	nStatusCode:	INT	:= 0;	// 0-OK, 1-Alarm, 2-Error

	
END_STRUCT
END_TYPE

// ---- DUTs/Structures/Coolers/T_CRYO_CRYOTELGT_CFG.TcDUT
TYPE T_CRYO_CRYOTELGT_CFG EXTENDS T_RS_BASE_CFG:
STRUCT

	tDelay_Read:		TIME 	:= T#150MS;	// Delay between sending each cmdList_Read[] command.
	nTimeoutState:		UDINT	:= 60000;	// 60 sec default timeout for starting and stopping cooler

	cmdList_Init:	ARRAY [1..8] OF T_CRYO_CRYOTELGT_CMD := [
		(cmd := 'VERSION', 				nReplies := 2),	// Current controller code version
		(cmd := 'MODE', 				nReplies := 2),	// MODE Cryocooler type, e.g. GT
		(cmd := 'SENSOR', 				nReplies := 2),	// Configured temp. sensor type, e.g. 'PT-100'
		(cmd := 'PWOUT=240', 			nReplies := 2),	// Set commanded power to 240 W
		(cmd := '', 					nReplies := 0),
		(cmd := '', 					nReplies := 0),
		(cmd := '', 					nReplies := 0),
		(cmd := '', 					nReplies := 0)];
	
	cmdList_Read:	ARRAY [1..16] OF T_CRYO_CRYOTELGT_CMD := [
		(cmd := 'ERROR', 				nReplies := 2),	// Controller error flags
		(cmd := 'COOLER', 				nReplies := 2),	// Cooler control mode, e.g. POWER or OFF
		(cmd := 'P', 					nReplies := 2),	// Measured cryocooler power
		(cmd := 'PWOUT', 				nReplies := 2),	// User commanded power
		(cmd := 'TC', 					nReplies := 2),	// Temperature sensor reading [K]
		(cmd := 'TEMP RJ', 				nReplies := 2),	// Reject temperature in [C]
		(cmd := '', 					nReplies := 0),
		(cmd := '', 					nReplies := 0),
		(cmd := '', 					nReplies := 0),
		(cmd := '', 					nReplies := 0),
		(cmd := '', 					nReplies := 0),
		(cmd := '', 					nReplies := 0),
		(cmd := '', 					nReplies := 0),
		(cmd := '', 					nReplies := 0),
		(cmd := '', 					nReplies := 0),
		(cmd := '', 					nReplies := 0)];
	

END_STRUCT
END_TYPE

// ---- DUTs/Structures/Coolers/T_CRYO_CRYOTELGT_CMD.TcDUT
TYPE T_CRYO_CRYOTELGT_CMD :
STRUCT
	cmd:		STRING	:= '';	// Command to send
	nReplies:	INT	:= 1;	// # of Replies
END_STRUCT
END_TYPE

// ---- DUTs/Structures/Coolers/T_CRYO_CRYOTELGT_CTRL.TcDUT
TYPE T_CRYO_CRYOTELGT_CTRL EXTENDS T_RS_BASE_CTRL:
STRUCT
	nDevCmd:	E_CRYO_CRYOTELGT_CMD := E_CRYO_CRYOTELGT_CMD.NONE;
	bStart:		BOOL;			// Control to Start/Stop the cooler.
	bPower:		BOOL;			// Update cooler power output.
	lrPower:	LREAL:= 240.0;	// Output power to set [W]
END_STRUCT
END_TYPE

// ---- DUTs/Structures/Coolers/T_CRYO_CRYOTELGT_STAT.TcDUT
TYPE T_CRYO_CRYOTELGT_STAT EXTENDS T_RS_BASE_STAT :
STRUCT
	
	nRetries:			UDINT := 0;			// Total number of retries in case of communication problems
	nDevState:			E_CRYO_CRYOTELGT_STATE := E_CRYO_CRYOTELGT_STATE.OFF;
	sDevState:			STRING := 'OFF';

	sReply:				STRING(255); 		(* Last Reply to predefined commands*)

	// Status attributes that are read from the controller via RS-232
	sVersion:			STRING;
	sMode:				STRING;
	sSensor:			STRING;
	sCtrlError:			STRING;
	sCtrlMode:			STRING;
	
	lrPowerMeasured:	LREAL;
	lrPowerCommanded:	LREAL;
	lrTempColdHead:		LREAL;
	lrTempReject:		LREAL;
	lrTempTarget:		LREAL;
	
	bPowerCmdActive:	BOOL;
	
END_STRUCT
END_TYPE

// ---- DUTs/Structures/Misc/T_CRYO_VOTE_LIST.TcDUT
// This structure is used to keep indexes of minimal reading differences
TYPE T_CRYO_VOTE_LIST :
STRUCT
	nIndex1:	INT;
	nIndex2:	INT;
	lrValue:	LREAL;	
END_STRUCT
END_TYPE

// ---- DUTs/Structures/Pumps/T_CRYO_PUMP_ATM2303M_CFG.TcDUT
TYPE T_CRYO_PUMP_ATM2303M_CFG EXTENDS T_CRYO_PUMP_SERIAL_CFG:
STRUCT
// TODO: Add specific configuration here

	// Definition of commands
	C_CMD_NONE:		STRING(16) := '';
	C_CMD_IDN:		STRING(16) := '#000IDN';
	C_CMD_RDI:		STRING(16) := '#000RDI';
	C_CMD_VER:		STRING(16) := '#000VER';
	C_CMD_DEF:		STRING(16) := '#000DEF';
	C_CMD_SEL:		STRING(16) := '#000SEL10';
	C_CMD_TIM:		STRING(16) := '#000TIM';
	C_CMD_STA:		STRING(16) := '#000STA';
	C_CMD_LEV:		STRING(16) := '#000LEV10';

END_STRUCT
END_TYPE

// ---- DUTs/Structures/Pumps/T_CRYO_PUMP_ATM2303M_STAT.TcDUT
TYPE T_CRYO_PUMP_ATM2303M_STAT EXTENDS T_CRYO_PUMP_BASE_STAT :
STRUCT

	// Digital status input signals
	bSpeed100:			BOOL;	// pump speed > 100 rpm
	
	
	// STA command
	// All attributes are defined in T_CRYO_PUMP_BASE_STAT
	
	// LEV10 command
	nNominalSpeed:				DINT;	// [rpm]
	nStandbySpeed:				DINT;	// [rpm]
	nSetPoint_AtSpeed:			DINT;	// ‘At speed’ relay set point (3 to 50%)
	nSetPoint_Temp:				DINT;	// temperature set point (30 to 65°C)
	nSetPoint_BearingWarn:		DINT;	// landing bearing warning set point (0 to 99%)
	nSetPoint_BearingCounter:	DINT;	// landing bearing counter (0 to 100%)
	
	// SEL command
	
	// VER Command (4 version strings)
	sVer1:	STRING;
	sVer2:	STRING;
	sVer3:	STRING;
	sVer4:	STRING;

	sIDN:	STRING;
	sRDI:	STRING;
	
	
END_STRUCT
END_TYPE

// ---- DUTs/Structures/Pumps/T_CRYO_PUMP_BASE_CFG.TcDUT
TYPE T_CRYO_PUMP_BASE_CFG EXTENDS T_RS_BASE_CFG:
STRUCT

	nModel:				DINT := 0;			// Model 0 indicates the base FB.
	nTimeoutState:		UDINT	:= 600000;	// 600 sec default timeout for starting and stopping pump
	

END_STRUCT
END_TYPE

// ---- DUTs/Structures/Pumps/T_CRYO_PUMP_BASE_CTRL.TcDUT
TYPE T_CRYO_PUMP_BASE_CTRL EXTENDS T_RS_BASE_CTRL:
STRUCT
	bStart:		BOOL;	// Control to Start/Stop the pump.
END_STRUCT
END_TYPE

// ---- DUTs/Structures/Pumps/T_CRYO_PUMP_BASE_STAT.TcDUT
TYPE T_CRYO_PUMP_BASE_STAT EXTENDS T_RS_BASE_STAT :
STRUCT
	
	nRetries:			UDINT := 0;			// Total number of retries in case of communication problems
	nPumpState:			E_CRYO_PUMP_STATE := E_CRYO_PUMP_STATE.OFF;
	sPumpState:			STRING := 'OFF';

	sReply:				STRING(255); 		(* Last Reply to predefined commands*)

	// Digital status input signals
	bReady:				BOOL;	// If TRUE, pump is operational
	bMoving:			BOOL;	// If TRUE, pump is rotating, i.e. speed > 0.
	bWarning:			BOOL;	// presence of a warning
	bAlarm:				BOOL;	// presence of an alarm
	
	// Values obtained via serial communication
	nCtrlMode:			DINT;	// e.g. 0-Hand held, 1-Remote, 2-Serial, etc
	sCtrlMode:			STRING;	// e.g. 'Hand held', 'Remote', 'Serial', etc

	bON:				BOOL;	// Flag if Motor Pump is ON
	nElecPower:			DINT;	// Electronic drive power [W]
	nElecHours:			DINT;	// Electronic drive unit operating hours
	nElecTemp:			DINT;	// Drive Electronics Temperature [degC]
	nMotorCurr:			DINT;	// Pump Motor Current [mA]
	nMotorVolt:			DINT;	// Pump Motor Voltage [V]
	nPumpHours:			DINT;	// Pump operating hours
	nPumpSpeed:			DINT;	// Pump Motor Speed [rpm]
	nPumpTemp:			DINT;	// Pump Temperature[degC]
	
	
	
END_STRUCT
END_TYPE

// ---- DUTs/Structures/Pumps/T_CRYO_PUMP_CMD.TcDUT
TYPE T_CRYO_PUMP_CMD :
STRUCT
	cmd:	STRING	:= '';	// Command to send
	length:	DINT	:= 1;	// Reply length
END_STRUCT
END_TYPE

// ---- DUTs/Structures/Pumps/T_CRYO_PUMP_HIPACE30_CFG.TcDUT
TYPE T_CRYO_PUMP_HIPACE30_CFG EXTENDS T_CRYO_PUMP_SERIAL_CFG:
STRUCT
// HIPACE30 specific command configuration.
// Pfeiffer Vacuum protocol for RS-485 interface.
// Assumed RS-485 device ID=1 (001) !!!

	// Definition of commands
	C_CMD_NONE:				STRING(16) := '';
	C_CMD_sCtrlViaInt:		STRING(16) := '0011006003001';	// Control via DIO
	C_CMD_sFwVersion:		STRING(16) := '0010031202=?';
	C_CMD_sHwVersion:		STRING(16) := '0010035402=?';
	C_CMD_nNominalSpeed:	STRING(16) := '0010039902=?';
	
	C_CMD_bON:				STRING(16) := '0010002302=?';
	C_CMD_nCtrlMode:		STRING(16) := '0010006002=?';
	C_CMD_sErrorCode:		STRING(16) := '0010030302=?';
	C_CMD_bTargetSpeed:		STRING(16) := '0010030602=?';
	C_CMD_nMotorCurr:		STRING(16) := '0010031002=?';
	C_CMD_nPumpHours:		STRING(16) := '0010031102=?';
	C_CMD_nMotorVolt:		STRING(16) := '0010031302=?';
	C_CMD_nElecHours:		STRING(16) := '0010031402=?';
	C_CMD_nElecTemp:		STRING(16) := '0010032602=?';
	C_CMD_nPumpTemp:		STRING(16) := '0010034602=?';
	C_CMD_nPumpSpeed:		STRING(16) := '0010039802=?';
	

END_STRUCT
END_TYPE

// ---- DUTs/Structures/Pumps/T_CRYO_PUMP_HIPACE30_STAT.TcDUT
TYPE T_CRYO_PUMP_HIPACE30_STAT EXTENDS T_CRYO_PUMP_BASE_STAT :
STRUCT

(*
Type:
0 - old bool: 0=FALSE, NOT 0 = TRUE.
1 - UDINT
2 - REAL * 100 (with leading zeros), e.g. 001571 corresponds with 15.71
4 - STRING (6)
7 - UINT (000 to 999)

INIT commands
023 MotorPump Motor pump 0 = off 1 = on 0 RW 0 1 1
060 CtrlViaInt Control via interface 7 RW 1 255 1
	1 = remote 
	2 = RS-485 
	4 = PV.can
	8 = Fieldbus
	16 = E74
	255 = unlock interface selection

312 Fw version Firmware version electronic drive unit 4 R
354 HW Version Hardware version electronic drive unit 4 R

STATUS commands
303 Error code Error code 4 R
306 SetSpdAtt Target speed reached 0 = no 1 = yes 0 R 0 1
310 DrvCurrent Drive current 2 R A 0 9999.99
311 OpHrsPump Operating hours pump 1 R h 0 65535
313 DrvVoltage Drive voltage 2 R V 0 9999.99
314 OpHrsElec Operating hours electronic drive unit 1 R h 0 65535
316 *** DrvPower Drive power 1 R W 0 999999
319 *** PumpCycles Pump cycles 1 R 0 65535
326 TempElec Temperature electronics 1 R °C 0 999999
346 ^^^ TempMotor Temperature motor 1 R °C 0 999999
397 *** SetRotSpd Set rotation speed (rpm) 1 R rpm 0 999999
398 ActualSpd Actual rotation speed (rpm) 1 R rpm 0 999999
399 NominalSpd Nominal rotation speed (rpm) 1 R rpm 0 999999

*)

// INIT commands
	sFwVersion:		STRING(8);
	sHwVersion:		STRING(8);

// STATUS commands
	sFailureCode:	STRING(8) := 'OK';
	bTargetSpeed:	BOOL;		// Target Speed Reached
	nNominalSpeed:	DINT;		// [rpm] Nominal Pump Speed
	lrMotorVolt:	LREAL;		// Pump Motor Voltage [V]
	
	bFailure:		BOOL := FALSE;	// Err of Wrn (see cmd 303)
END_STRUCT
END_TYPE

// ---- DUTs/Structures/Pumps/T_CRYO_PUMP_MODBUS_CFG.TcDUT
TYPE T_CRYO_PUMP_MODBUS_CFG EXTENDS T_CRYO_PUMP_BASE_CFG:
STRUCT
	nSlaveID:	BYTE := 1;
	nVersion:	E_ECODRY_VERSION;
	
	// Register Addresses. See M_UserConfigure().
	aAddr:		ARRAY [1..8] OF INT := [0, 0, 0, 0, 0, 0, 0, 0];
	aWords:		ARRAY [1..8] OF INT := [0, 0, 0, 0, 0, 0, 0, 0];
	
END_STRUCT
END_TYPE

// ---- DUTs/Structures/Pumps/T_CRYO_PUMP_MODBUS_CTRL.TcDUT
TYPE T_CRYO_PUMP_MODBUS_CTRL EXTENDS T_CRYO_PUMP_BASE_CTRL:
STRUCT
	nCmdType:	DINT	:= E_MODBUS_CMD_TYPE.READ;	// Command type; 0-Read, 1-Write
	nRegister:	DINT;								// Command register
	nWords:		DINT	:= 1;						// Number of words
	nValue:		DINT;								// Parameter value
END_STRUCT
END_TYPE

// ---- DUTs/Structures/Pumps/T_CRYO_PUMP_MODBUS_STAT.TcDUT
TYPE T_CRYO_PUMP_MODBUS_STAT EXTENDS T_CRYO_PUMP_BASE_STAT:
STRUCT
	nInputBuffer: 			ARRAY [0..300] OF BYTE;	// Binary data read from ECODRY
	
	lrFreqRef:				LREAL;	// Frequency Reference 0x0040
	lrOutFreq:				LREAL;	// Output Frequency 0x0041
//	lrOutCurrent:			LREAL;	// Output Current 0x0042
	lrOutVoltRef:			LREAL;	// Output Voltage Reference 0x0045
//	lrDcBusVolt:			LREAL;	// DC Bus Voltage 0x0046
	lrOutPower:				LREAL;	// Output Power 0x0047
//	lrTemperature:			LREAL;	// Heatsink Temperature 0x0068

	nSwFlash:				UINT;	// Software No. (Flash) 0x004D
	nSwRom:					UINT;	// Software No. (ROM) 0x005B
	nOpTime:				UINT;	// Accumulated Operation Time 0x004C
	nNumRunCmd:				UINT;	// Number of Run Commands 0x0075
	nFanOpTime:				UINT;	// Cooling Fan Operation Time  0x0067
	
	nServiceHours:			UINT;	// Service Hours 0x0667
	nNumPumpDowns:			UINT;	// Pump-down Cycles after Service 0x0669
	nDaysUntilService:		UINT;	// Days before Service 0x066C

END_STRUCT
END_TYPE

// ---- DUTs/Structures/Pumps/T_CRYO_PUMP_MVP030_CFG.TcDUT
TYPE T_CRYO_PUMP_MVP030_CFG EXTENDS T_CRYO_PUMP_SERIAL_CFG:
STRUCT
// MVP030 specific command configuration.
// Pfeiffer Vacuum protocol for RS-485 interface.
// Assumed RS-485 device ID=1 (001) !!!

	// Definition of commands
	C_CMD_NONE:				STRING(16) := '';
	C_CMD_sCtrlViaInt:		STRING(16) := '0011006003001';	// Control via DIO
	C_CMD_sFwVersion:		STRING(16) := '0010031202=?';
	C_CMD_sHwVersion:		STRING(16) := '0010035402=?';
	C_CMD_nNominalSpeed:	STRING(16) := '0010039902=?';
	
	C_CMD_bON:				STRING(16) := '0010001002=?';
	C_CMD_nCtrlMode:		STRING(16) := '0010006002=?';
	C_CMD_sErrorCode:		STRING(16) := '0010030302=?';
	C_CMD_nMotorCurr:		STRING(16) := '0010031002=?';
	C_CMD_nPumpHours:		STRING(16) := '0010031102=?';
	C_CMD_nMotorVolt:		STRING(16) := '0010031302=?';
	C_CMD_nElecPower:		STRING(16) := '0010031602=?';
	C_CMD_nPumpTemp:		STRING(16) := '0010033002=?';
	C_CMD_nPumpSpeed:		STRING(16) := '0010039802=?';
	
	C_CMD_sID000:			STRING(16) := '0001079706000001';	// Change all IDs to 1

END_STRUCT
END_TYPE

// ---- DUTs/Structures/Pumps/T_CRYO_PUMP_MVP030_STAT.TcDUT
TYPE T_CRYO_PUMP_MVP030_STAT EXTENDS T_CRYO_PUMP_BASE_STAT :
STRUCT

(*
Type:
0 - old bool: 0=FALSE, NOT 0 = TRUE.
1 - UDINT
2 - REAL * 100 (with leading zeros), e.g. 001571 corresponds with 15.71
4 - STRING (6)
7 - UINT (000 to 999)

INIT commands
312 Fw version Firmware version electronic drive unit 4 R
354 HW Version Hardware version electronic drive unit 4 R
399 NominalSpd Nominal rotation speed (rpm) 1 R rpm 0 999999

STATUS commands
010 Pumpg-Statn Pump 0 = off 1 = on 0 RW 0 1 0 x
060 CtrlViaInt Operation of the interface 
	1 = remote
	2 = RS-485
	4 = PV.can
	32 = Keys on the front panel

303 Error code Error code 4 R
	Err098 Internal communication error between interface board and drive
	Err117 Vacuum pump excess temperature (> 90 °C)
	Err174 Vacuum pump blocked
	Wrn117 High temperature vacuum pump (> 75 °C)

310 DrvCurrent Drive current 2 R A 0 9999.99
311 OpHrsPump Operating hours pump 1 R h 0 65535
313 DrvVoltage Drive voltage 2 R V 0 9999.99
316 *** DrvPower Drive power 1 R W 0 999999
330 TempPump Pump temperature 1 R °C 0 999999
398 ActualSpd Actual rotation speed (rpm) 1 R rpm 0 999999

*)

// INIT commands
	sFwVersion:		STRING(8);
	sHwVersion:		STRING(8);

// STATUS commands
	sFailureCode:	STRING(8) := 'OK';
	bTargetSpeed:	BOOL;		// Target Speed Reached
	nNominalSpeed:	DINT;		// [rpm] Nominal Pump Speed
	lrMotorVolt:	LREAL;		// Pump Motor Voltage [V]

	
	bFailure:		BOOL := FALSE;	// Err of Wrn (see cmd 303)
END_STRUCT
END_TYPE

// ---- DUTs/Structures/Pumps/T_CRYO_PUMP_SERIAL_CFG.TcDUT
TYPE T_CRYO_PUMP_SERIAL_CFG EXTENDS T_CRYO_PUMP_BASE_CFG:
STRUCT
	//
	// List of INIT commands.
	//
	cmdList_Init:	ARRAY [1..8] OF T_CRYO_PUMP_CMD;

	//
	//	List of READ (and WRITE) commands.
	// NOTE: Monitoring loop stops on first cmd = ''.
	//
	cmdList_Read:	ARRAY [1..16] OF T_CRYO_PUMP_CMD;

END_STRUCT
END_TYPE

// ---- DUTs/Structures/Sensors/T_CRYO_IOLINK_SENSOR_STATUS.TcDUT
TYPE T_CRYO_IOLINK_SENSOR_STATUS :
STRUCT
	bInRange:			BOOL;
	bUnderrange:		BOOL;
	bOverrange:			BOOL;
	bError:				BOOL;
	bValid:				BOOL;
	
	lrValue:			LREAL;		// Reading in UU
	
	sUnits:				STRING(16);
	sType:				STRING(32);	// Sensor type, e.g. 'Flow' or 'Temperature'.
	sStatus:			STRING	:= 'OK';

END_STRUCT
END_TYPE

// ---- DUTs/Structures/Sensors/T_CRYO_PRESSURE_STATUS.TcDUT
TYPE T_CRYO_PRESSURE_STATUS :
STRUCT
	bInRange:		BOOL	:= FALSE;
	bValid:			BOOL	:= FALSE;
	bWarningSens1:	BOOL	:= TRUE;
	bWarningSens2:	BOOL	:= TRUE;
	bInVacuum:		BOOL	:= FALSE;
	bVacuumGood:	BOOL	:= FALSE;
	lrPressure:		LREAL;	// Pressure [mbar]
END_STRUCT
END_TYPE

// ---- DUTs/Structures/Sensors/T_CRYO_PRESSURE_VOTE_STATUS.TcDUT
TYPE T_CRYO_PRESSURE_VOTE_STATUS :
STRUCT
	bSimulated:		BOOL;				// Flag indicating if the value is simulated.
	lrSimPressure:	LREAL;				// Simulated pressure value [mbar]

	bValid:			BOOL	:= FALSE;	// Flag indicating if the value is valid.
	lrPressure:		LREAL;				// Calculated Pressure [mbar]
	sStatus:		STRING;				// Status string

	// Flags indicating warnings for each connected sensor.
	// Only connected sensors can have warnings!!!
	bWarnSens1:		BOOL	:= TRUE;
	bWarnSens2:		BOOL	:= TRUE;
	bWarnSens3:		BOOL	:= TRUE;
	bWarnSens4:		BOOL	:= TRUE;
	bWarnSens5:		BOOL	:= TRUE;

	// Flags for each sensor indicating if it is connected.
	bConnSens1:		BOOL	:= FALSE;
	bConnSens2:		BOOL	:= FALSE;
	bConnSens3:		BOOL	:= FALSE;
	bConnSens4:		BOOL	:= FALSE;
	bConnSens5:		BOOL	:= FALSE;
END_STRUCT
END_TYPE

// ---- DUTs/Structures/Sensors/T_CRYO_PT100_OHM2C_REC.TcDUT
TYPE T_CRYO_PT100_OHM2C_REC :
STRUCT
	celsius:	LREAL;	// Temperature in celsius [C]
	ohm:		LREAL;	// Resistance in [Ohm]
END_STRUCT
END_TYPE

// ---- DUTs/Structures/Sensors/T_CRYO_SBG232_STAT.TcDUT
TYPE T_CRYO_SBG232_STAT :
STRUCT
	bConfigured:	BOOL;
	sName:			STRING;
	sStatus:		STRING	:= 'OK';
	
	flow:	T_CRYO_IOLINK_SENSOR_STATUS;	// Flow status
	temp:	T_CRYO_IOLINK_SENSOR_STATUS;	// Temperature status
END_STRUCT
END_TYPE

// ---- DUTs/Structures/Sensors/T_CRYO_SENSOR_STATUS.TcDUT
TYPE T_CRYO_SENSOR_STATUS :
STRUCT
	//
	// Status coming from the analog input terminal.
	// This is nothing to do with the sensor, i.e. the reading can be
	// inside the input terminal measuring range but still it might
	// not be inside the sensor measuring range!
	//
	bInputUnder:		BOOL;
	bInputOver:			BOOL;
	bInputError:		BOOL;
	bInputToggle:		BOOL;
	bInputValid:		BOOL;
	bInputActive:		BOOL	:= FALSE;
	nRawValue:			INT;

	// Calculated status of the sensor
	bError:				BOOL;
	bValid:				BOOL;

END_STRUCT
END_TYPE

// ---- DUTs/Structures/Sensors/T_CRYO_SENSOR_STATUS_PRESS.TcDUT
TYPE T_CRYO_SENSOR_STATUS_PRESS EXTENDS T_CRYO_SENSOR_STATUS :
STRUCT
	nType:		E_CRYO_SENSOR_TYPE_PRESS;

	// Measured and calculated values
	lrVoltage:		LREAL;	// Voltage [V]
	lrPressure:		LREAL;	// Pressure [mbar]

	// Status coming from the user evaluation.
	// These flags indicate if the reading is outside the sensor operational range.
	// Therefore, the voltage might be correctly measured but
	// the pressure is outside what the sensor can measure.	
	bValueInRange:		BOOL;	// Flag if reading is inside SENSOR(!) range
	bValueOverrange:	BOOL;	// Flag if reading is outside SENSOR(!) range
	bValueUnderrange:	BOOL;	// Flag if reading is outside SENSOR(!) range

END_STRUCT
END_TYPE

// ---- DUTs/Structures/Sensors/T_CRYO_SENSOR_STATUS_TEMP.TcDUT
TYPE T_CRYO_SENSOR_STATUS_TEMP EXTENDS T_CRYO_SENSOR_STATUS :
STRUCT
	nType:		E_CRYO_SENSOR_TYPE_TEMP;
	
	lrRamp:		LREAL;	// Temperature ramp [deg/min]
	lrTempC:	LREAL;	// Temperature in deg C
	lrTempK:	LREAL;	// Temperature in deg K
END_STRUCT
END_TYPE

// ---- DUTs/Structures/Sensors/T_CRYO_TEMPERATURE_STATUS.TcDUT
TYPE T_CRYO_TEMPERATURE_STATUS :
STRUCT
	bSimulated:		BOOL;				// Flag indicating if the value is simulated.
	lrSimTempK:		LREAL;				// Simulated temperature value in [K].

	bInRange:		BOOL	:= FALSE;
	bValid:			BOOL	:= FALSE;
	bWarningSens1:	BOOL	:= TRUE;
	bWarningSens2:	BOOL	:= TRUE;
	lrRamp:			LREAL;				// Temperature ramp [deg/min]
	lrTempC:		LREAL;				// Temp [deg C]
	lrTempK:		LREAL;				// Temp [deg K]
END_STRUCT
END_TYPE

// ---- DUTs/Structures/Subsystems/Evacuation/T_CRYO_EVACUATION_SYSTEM_STATUS.TcDUT
TYPE T_CRYO_EVACUATION_SYSTEM_STATUS :
STRUCT
	bDone:			BOOL;			// Flag if controller is OK
	bBusy:			BOOL;			// Flag if controller is BUSY
	bEnabled:		BOOL := FALSE;	// Controller active while bEnable is TRUE
	bError:			BOOL;			// Flag if controller is OK
	bActive:		BOOL;			// Flag if controller is ACTIVE
	bEmergency:		BOOL := FALSE;	// Flag if there was Emergency valve closure
	bRootPumpON:	BOOL;			// Flag if Root Pump is running
	bTurboPumpON:	BOOL;			// Flag if Turbo Pump is running
	bTurboPump10min:BOOL;			// Flag if Turbo Pump has been running for more than 10 min
	bValveOpen:		BOOL;			// Flag if Evacuation Valve is open

	// Generic controller OK flag.
	// Used for problems other than from the actuator.
	// This flag is used for problems coming from controllers
	// that extend the functionality of FB_CRYO_BIN_CTRL.
	bCtrlOK:	BOOL := TRUE;		

	nCycleCounter:	UDINT := 0;
	nLastCommand:	E_CRYO_BIN_ACT_CMD	:= E_CRYO_BIN_ACT_CMD.NONE;	// Command
	nState:			E_CRYO_EVAC_SYS_STATE	:= E_CRYO_EVAC_SYS_STATE.NONE;
	
	sState:			STRING(64);		// State as text
	sStatus:		STRING(64);		// Status as text
END_STRUCT
END_TYPE

// ---- DUTs/Structures/Subsystems/Evacuation/T_CRYO_EVAC_CFG.TcDUT
TYPE T_CRYO_EVAC_CFG :
STRUCT
	nPressGaugeType1:	E_CRYO_SENSOR_TYPE_PRESS := E_CRYO_SENSOR_TYPE_PRESS.PKR_360;
	nPressGaugeType2:	E_CRYO_SENSOR_TYPE_PRESS := E_CRYO_SENSOR_TYPE_PRESS.PKR_360;

	bPressSimulation:	BOOL := FALSE;	// Flag is pre-vacuum pressure is simulated.

	lrThld_Prevac:					LREAL := 0.005;	// Prevacuum pressure threshold
	lrThld_PrevacHigh:				LREAL := 5.0;	// Prevacuum pressure too high threshold
	// Cryo pressure threshold for safe Turbo Pump start
	lrThld_TP_SafeStartPressure:	LREAL := 0.01;	
	// Cryo pressure threshold for safe Valve opening
	lrThld_Valve_SafeOpenPressure:	LREAL := 0.1;	
	
	tDelay:		TIME := T#3S;	// Time delay before stopping Turbo Pump
END_STRUCT
END_TYPE

// ---- DUTs/Structures/Subsystems/Evacuation/T_CRYO_EVAC_CFG_50000.TcDUT
TYPE T_CRYO_EVAC_CFG_50000 :
STRUCT
	// Pressure sensor gauge types
	nType_VAG1:		E_CRYO_SENSOR_TYPE_PRESS := E_CRYO_SENSOR_TYPE_PRESS.PKR_360;
	nType_VAG2:		E_CRYO_SENSOR_TYPE_PRESS := E_CRYO_SENSOR_TYPE_PRESS.PKR_360;
	nType_VAG3:		E_CRYO_SENSOR_TYPE_PRESS := E_CRYO_SENSOR_TYPE_PRESS.PKR_360;
	nType_VAGF1:	E_CRYO_SENSOR_TYPE_PRESS := E_CRYO_SENSOR_TYPE_PRESS.PKR_360;
	nType_VAGF2:	E_CRYO_SENSOR_TYPE_PRESS := E_CRYO_SENSOR_TYPE_PRESS.PKR_360;
	nType_VAGG1:	E_CRYO_SENSOR_TYPE_PRESS := E_CRYO_SENSOR_TYPE_PRESS.PKR_360;
	nType_VAGG2:	E_CRYO_SENSOR_TYPE_PRESS := E_CRYO_SENSOR_TYPE_PRESS.PKR_360;

	// Flag is pressures are simulated.
	// TODO: Define individual flags for each sensor.
	bPressSimulation:	BOOL := FALSE;	

	lrThld_Prevac:			LREAL := 0.1;	// Prevacuum pressure threshold [mbar] 
	lrThld_PrevacHigh:		LREAL := 5.0;	// Prevacuum pressure too high threshold [mbar]
	lrThld_Vacuum:			LREAL := 0.0001;// At this Cryo pressure evacuation has started [mbar]
	
	tDelay:		TIME := T#3S;	// Delay after closing all valves before stopping Pumps
END_STRUCT
END_TYPE

// ---- DUTs/Structures/Subsystems/Evacuation/T_CRYO_EVAC_CTRL.TcDUT
TYPE T_CRYO_EVAC_CTRL :
STRUCT
	bEnable_RP:		BOOL := FALSE;
	bEnable_TP:		BOOL := FALSE;
	bEnable_Valve:	BOOL := FALSE;
END_STRUCT
END_TYPE

// ---- DUTs/Structures/Subsystems/Evacuation/T_CRYO_EVAC_CTRL_50000.TcDUT
TYPE T_CRYO_EVAC_CTRL_50000 :
STRUCT
	// Flags for control of pumps.
	// Seeting the flag to TRUE  will start the pump.
	// Seeting the flag to FALSE will stop  the pump.
	bEnable_PVP:	BOOL := FALSE;	// Prevacuum pump
	bEnable_TMP:	BOOL := FALSE;	// Turbo molecular pump
	
	// Flags for control of valves
	// Seeting the flag to TRUE  will open  the valve.
	// Seeting the flag to FALSE will close the valve.
	bEnable_PVV1:	BOOL := FALSE;
	bEnable_PVV2:	BOOL := FALSE;
	bEnable_PVV3:	BOOL := FALSE;
	bEnable_PVV4:	BOOL := FALSE;
	bEnable_GBV:	BOOL := FALSE;
	
END_STRUCT
END_TYPE

// ---- DUTs/Structures/Subsystems/Evacuation/T_CRYO_EVAC_STAT.TcDUT
TYPE T_CRYO_EVAC_STAT :
STRUCT
	bEnabled:		BOOL := FALSE;	// Controller active while bEnable is TRUE
	bConfigured:	BOOL := FALSE;	// Flag if controller has been configured.
	bError:			BOOL;			// Flag if controller is OK
	bActive:		BOOL;			// Flag if controller is ACTIVE
	bEmergency:		BOOL := FALSE;	// Flag if there was Emergency valve closure
	bRootPumpON:	BOOL;			// Flag if Root Pump is running
	bTurboPumpON:	BOOL;			// Flag if Turbo Pump is running
	bValveOpen:		BOOL;			// Flag if Evacuation Valve is open
	bValveAfterTP:	BOOL := FALSE;	// Flag if Evacuation Valve should open after TP has started

	// Generic controller OK flag.
	// Used for problems other than from the actuator.
	// This flag is used for problems coming from controllers
	// that extend the functionality of FB_CRYO_BIN_CTRL.
	bCtrlOK:	BOOL := TRUE;		

	nCycleCounter:	UDINT := 0;
	nState:			E_CRYO_EVAC_STATE	:= E_CRYO_EVAC_STATE.NONE;
	
	sErrorText:		STRING(64);		// Error as text
	sState:			STRING(64);		// State as text
	sStatus:		STRING(64);		// Status as text
END_STRUCT
END_TYPE

// ---- DUTs/Structures/Subsystems/Evacuation/T_CRYO_EVAC_STAT_50000.TcDUT
TYPE T_CRYO_EVAC_STAT_50000 :
STRUCT
	bEnabled:		BOOL := FALSE;	// Controller active while bEnable is TRUE
	bConfigured:	BOOL := FALSE;	// Flag if controller has been configured.
	bError:			BOOL;			// Flag if controller is OK
	bActive:		BOOL;			// Flag if controller is ACTIVE
	bEmergency:		BOOL := FALSE;	// Flag if there was Emergency valve closure
	bRootPumpON:	BOOL;			// Flag if Root Pump is running
	bTurboPumpON:	BOOL;			// Flag if Turbo Pump is running

	// Generic controller OK flag.
	// Used for problems other than from the actuator.
	// This flag is used for problems coming from controllers
	// that extend the functionality of FB_CRYO_BIN_CTRL.
	bCtrlOK:	BOOL := TRUE;		

	nCycleCounter:	UDINT := 0;
	nState:			E_CRYO_EVAC_STATE_50000	:= E_CRYO_EVAC_STATE_50000.NONE;
	
	sErrorText:		STRING(64);		// Error as text
	sState:			STRING(64);		// State as text
	sStatus:		STRING(64);		// Status as text
END_STRUCT
END_TYPE

// ---- DUTs/Structures/Subsystems/Evacuation/T_CRYO_EVAC_SYS_INPUT.TcDUT
// NOTE: Not used yet !!!
// Should replace input parameters of FB_CRYO_EVACUATION_SYSTEM.
// Should be set with NEW method FB_CRYO_CTRL::M_SetEvacSystemInputData().
TYPE T_CRYO_EVAC_SYS_INPUT :
STRUCT
	//
	// System configuration
	//
	// Time between closing Vac valve and Switching OFF the vac Pump [ms]
	nTime_DeltaTValve:		UDINT;	
	// Time [ms] to run Turbo Pump to consider vacuum is good (useful when cryostat is cold)
	nTime_TurboPump:		UDINT;	

	lrPress_Atm:			LREAL;	// Atmospheric pressure limit   [mbar]

	lrTemp_Precooled:		LREAL;	// Precooled temperature limit [K]
	lrTemp_Warm:			LREAL;	// Warm      temperature limit [K]

	//
	// System configuration
	//
	lrTemp_Cryo:			T_CRYO_TEMPERATURE_STATUS;	// Cold Bench temperature	
	lrPressure_Cryo:		T_CRYO_PRESSURE_STATUS;		// Cryostat Pressure
	lrPressure_Evac:		T_CRYO_PRESSURE_STATUS;		// Evacuation Pressure
	bRepressValveOpen:		BOOL;	// Repressure Valve Open flag
	bRepressValveOK:		BOOL;	// Repressure Valve OK flag
END_STRUCT
END_TYPE

// ---- DUTs/Structures/System/T_CRYO_CFG.TcDUT
TYPE T_CRYO_CFG :
STRUCT
	lrTemp_Precooled:		LREAL := 110.0;	// Precooled temperature limit [K]
	lrTemp_Cold:			LREAL :=  80.0;	// Cool      temperature limit [K]
	lrTemp_Warm:			LREAL := 283.15;// Warm      temperature limit [K] = 10 C
	
	// Delat-T SetPoint between Detector and Coldbench during WarmUp
	lrTemp_DeltaDet_Bench_Low:	LREAL	:= 10.0;
	// Delat-T SetPoint between Detector and Coldbench during WarmUp	
	lrTemp_DeltaDet_Bench_High:	LREAL	:= 5.0;		

	lrTemp_LN2ValveOpen:	LREAL := 91.27;		// Open  valve if temperature above this value [K]
	lrTemp_LN2ValveClose:	LREAL := 79.148;	// Close valve if temperature below this value [K]

	lrPress_Atm:			LREAL := 700.0;		// Atmospheric pressure limit   [mbar]
	lrPress_InVac:			LREAL := 10.0E-1;	// In vacuum limit   [mbar]
	lrPress_GoodVac:		LREAL := 10.0E-4;	// Good Vacuum limit [mbar]
	
	
	// Time between closing Vac valve and Switching OFF the vac Pump [ms]
	nTime_DeltaTValve:		UDINT := 2000;	
	// Vacuum Pump Settling Time [ms]
	nTime_VacPumpSettling:	UDINT := 1000;	
	// 10 min (600000ms) run of Turbo Pump to consider vac is good (useful when cryostat is cold)
	nTime_TurboPump:		UDINT := 600000;	
	
	//
	// Lakeshore 340 configuration
	//
	LS_CTRL_MODE:			INT		:= 2;		// Remote without local lock
	
	// Warm
	LS_W_PID_A_P:			UINT	:= 10;		// Warm state P controler value
	LS_W_PID_A_I:			UINT	:= 50;		// Warm state I controler value
	LS_W_PID_A_D:			UINT	:= 12;		// Warm state D controler value
	LS_W_Heater_Range:		UINT	:= 4;		// Warm Resistance power range
	LS_W_CTRL_RAMP:			LREAL	:= 1.0;		// Warm-up delta-T Kelvin per minutes
	LS_W_SETPOINT_A:		LREAL	:= 293.15;	// 20 Deg Celcius

	// Cold
	LS_C_PID_A_P:			UINT	:= 50;		// Cold state P controler value
	LS_C_PID_A_I:			UINT	:= 71;		// Cold state I controler value
	LS_C_PID_A_D:			UINT	:= 10;		// Cold state D controler value
	LS_C_Heater_Range:		UINT	:= 4;		// Cold Resistance power range
	LS_C_CTRL_RAMP:			LREAL	:= 0.0;		// Cooldown/Cooling delta-T Kelvin per minutes
	LS_C_SETPOINT_A:		LREAL	:= 40.0;	// -193,15 Deg Celcius

END_STRUCT
END_TYPE

// ---- DUTs/Structures/System/T_CRYO_CTRL.TcDUT
TYPE T_CRYO_CTRL :
STRUCT
	bExecute:	BOOL := FALSE;
	nCommand:	E_CRYO_CTRL_CMD := E_CRYO_CTRL_CMD.NONE;
	
	bReset:		BOOL := FALSE;		// RESET Command

	bEnable_Evac:		BOOL := FALSE;
	bEnable_Heater:		BOOL := FALSE;
	bEnable_Precool:	BOOL := FALSE;
	bEnable_Cool:		BOOL := FALSE;
	bEnable_Warmup:		BOOL := FALSE;
	bEnable_CCC:		BOOL := FALSE;
	bEnable_RepressSys:	BOOL := FALSE;
	bEnable_RepressCtrl:BOOL := FALSE;

	// Safe flags
	bSafe_Precool:		BOOL := FALSE;
	bSafe_Cooling:		BOOL := FALSE;
	bSafe_Warmup:		BOOL := FALSE;
	bSafe_Repress:		BOOL := FALSE;
	
	// Ignore underrange flags.
	// We know that the ColdBench PT100 is broken and gives -200 C.
	bIgnoreUnderrange_ColdBench:	BOOL := FALSE;
	
	// Lakeshore related control parameters
	bLS_UpdateSETP:		BOOL := FALSE;	// If TRUE, this flag will trigger Lakeshore SETP.
	lrLS_SETP:			LREAL := 40.0;	// New SETP
	lrLS_RAMP:			LREAL := 0.5;	// RAMP [K/min]
	
END_STRUCT
END_TYPE

// ---- DUTs/Structures/System/T_CRYO_LOG.TcDUT
// Last ten system logs
TYPE T_CRYO_LOG :
STRUCT
	// This could have been done much simpler as:
	// 	sLog: ARRAY [0..9] OF STRING(80);
	// However, this would make it hard to view individual strings
	// with OPC UA Clients.
	// That's why we use 'ptrLog[0..9]' to scroll through the strings.
	// See M_Configure() for how pointers are set.
	
	s0:		STRING(80);
	s1:		STRING(80);
	s2:		STRING(80);
	s3:		STRING(80);
	s4:		STRING(80);
	s5:		STRING(80);
	s6:		STRING(80);
	s7:		STRING(80);
	s8:		STRING(80);
	s9:		STRING(80);
END_STRUCT
END_TYPE

// ---- DUTs/Structures/System/T_CRYO_STAT.TcDUT
TYPE T_CRYO_STAT :
STRUCT
	bConfigured:	BOOL := FALSE;

	bDone:			BOOL;			// Flag if controller is OK
	bBusy:			BOOL;			// Flag if controller is BUSY
	bError:			BOOL;			// Flag if controller is OK
	bActive:		BOOL;			// Flag if controller is ACTIVE
	// Generic controller OK flag.
	// Used for problems other than from the actuator.
	// This flag is used for problems coming from controllers
	// that extend the functionality of FB_CRYO_BIN_CTRL.
	bCtrlOK:		BOOL := TRUE;		

	bInVacuum:		BOOL := FALSE;		
	bGoodVacuum:	BOOL := FALSE;		

	bHighestTempValid:	BOOL := FALSE;	// Highest temperature Valid flag
	bLowestTempValid:	BOOL := FALSE;	// Lowest temperature Valid flag
	bDiffTempValid:		BOOL := FALSE;	// TRUE if Temperature difference is Valid

	lrHighestTempK:	LREAL;	// Highest temperature [K] in Cryostat
	lrLowestTempK:	LREAL;	// Lowest temperature [K] in Cryostat
	lrDiffTempK:	LREAL;	// Temperature difference (DET -Lowest temperature) [K]
	lrLS_Power:		LREAL;	// Lakeshore Power Output [%]
	
	nCycleCounter:	UDINT := 0;
	nLastCommand:	E_CRYO_CTRL_CMD 	:= E_CRYO_CTRL_CMD.NONE;
	nState:			E_CRYO_CTRL_STATE	:= E_CRYO_CTRL_STATE.NONE;
	
	
	sState:			STRING(64);		// State as text

END_STRUCT
END_TYPE

// ---- POUs/MAIN.TcPOU
PROGRAM MAIN
VAR
	
	
	{attribute 'OPC.UA.DA' := '1'}
	Cryo_Ctrl:	FB_CRYO_CTRL;
	
	
	{attribute 'OPC.UA.DA' := '1'}
	SIM_Cryo_Ctrl:	FB_CRYO_SIM_CTRL;
	
	//
	// Pressure voting system testing
	//
	P1_1:	FB_CRYO_SENSOR_PRESSURE;
	P1_2:	FB_CRYO_SENSOR_PRESSURE;
	P1_3:	FB_CRYO_SENSOR_PRESSURE;
	P1_4:	FB_CRYO_SENSOR_PRESSURE;
	P1_5:	FB_CRYO_SENSOR_PRESSURE;
	P1:		FB_CRYO_PRESSURE_VOTE;	// Voting of P1_1..P1_5

	nVoteMethod:		E_CRYO_VOTE	:=E_CRYO_VOTE.V_3oo5;
	bP1_Sim:			BOOL := FALSE;
	SIM_Pressure_P1:	FB_CRYO_SIM_PRESSURE;		// P1 Pressure simulator
	pressOR_P1:			FB_CRYO_CMD_OVERRIDE;

	////////////////////////////
	// Temperature testing
	//
	T1:		FB_CRYO_SENSOR_TEMPERATURE;
	T2:		FB_CRYO_TEMPERATURE;
	nRampPeriodSec:		UDINT := 60;	// Ramp measurement period [sec]. Default 60 sec.
	tempOR_T2:	FB_CRYO_CMD_OVERRIDE;
	simT2:		BOOL;
	////////////////////////////
	
	
	//////////////////////////////////////////////////////////////////
	
	//
	// Threshold testing
	//
	thld1:		FB_CRYO_THLD_BASE;	// Threshold handling
	
	// Threshold levels in format
	// [<alarm low>, <warning low>, <warning high>, <alarm high>]
	aThlds:		ARRAY [1..4] OF LREAL	:= [-80.0, -60.0, 40.0, 80.0];
	aThldDelay:	ARRAY [1..4] OF UDINT	:= [1000, 0, 2000, 0];
	nThldMode:	E_CRYO_THLD_MODE := E_CRYO_THLD_MODE.FIXED;	// Threshold check mode
	lrHyst:		LREAL	:= 10.0;	// Threshold hysteresis
	lrThldRef:	LREAL	:= 0.0;		// Threshold reference for User defined active thresholds
	
	SIM_thld1:	FB_CRYO_SIM_SINE;	// Simulated signal for threshold testing
	SIM_thld2:	FB_CRYO_SIM_SINE;	// Simulated signal for threshold testing
	nSimPer1:	UDINT := 60000;		// Period [ms] of simulated sine curve #1
	nSimPer2:	UDINT := 16000;		// Period [ms] of simulated sine curve #2
	
	/////////////////////////////////////////////////////////////////////////
	/////////////////////////////////////////////////////////////////////////

	///////////////////
	// Lakeshore 336
	///////////////////
	// Lakeshore 336 (Ethernet interface)
	{attribute 'OPC.UA.DA' := '1'}
	LS336_TCP:		FB_LAKESHORE_TCP;		// LakeShore based on FB_TCP_CLIENT



///////////////////////////////////////////////////////////////////
// Pumps and evacuations
///////////////////////////////////////////////////////////////////
	
	evac_pds:	FB_CRYO_EVAC_PDS;

	evac_lab:	FB_CRYO_EVAC_ECODRY_ATH2303M;	
	
	evac_micado:	FB_CRYO_EVAC_MICADO;

	// Cryostat pressure (sensor and evaluation)
	cryo_lab_press1:	FB_CRYO_SENSOR_PRESSURE;	// Cryostat pressure gauge #1
	cryo_lab_pressure:	FB_CRYO_PRESSURE_VOTE;		// Cryostat pressure 
	
	// Flags to control start/stop of pumps
	bEnable_evac_pds:	BOOL;
	bEnable_evac_lab:	BOOL;
	bEnable_evac_mic:	BOOL;
	
	// Simulation flags
	bSim_cryo_lab_pressure:	BOOL;
	
	
	//////////////////////////////
	// SUNPOWER Cryotel GT Cooler
	//////////////////////////////
	cooler:			FB_CRYO_CRYOTELGT;
	bEnable_cooler:	BOOL;
	
	
	///////////////////
	// MICADO
	///////////////////
	sensor_VAGF1:	FB_CRYO_SENSOR_PRESSURE;	// Cryo pressure gauge VAG F1
	sensor_VAGF2:	FB_CRYO_SENSOR_PRESSURE;	// Cryo pressure gauge VAG F2
	sensor_VAGG1:	FB_CRYO_SENSOR_PRESSURE;	// Cryo pressure gauge VAG G1
	sensor_VAGG2:	FB_CRYO_SENSOR_PRESSURE;	// Cryo pressure gauge VAG G2
	VAGF:	FB_CRYO_PRESSURE_VOTE;				// Cryo pressure F
	VAGG:	FB_CRYO_PRESSURE_VOTE;				// Cryo pressure G

	// Valve Command handling
	cmdPVV1:	FB_CRYO_ACTUATOR_CMD;
	bCmdPVV1:	BOOL;	// Open/Close command for PVV1
	bIntlkPVV1:	BOOL;	// Interlock for PVV1
	
	///////////////////
	// Simulation
	/////////////////
	
	mic_valves:	FB_SIM_MICADO_VALVES;
	mic_pumps:	FB_SIM_MICADO_PUMPS;
	
	// Pressure values
	q_nVAG1		AT %Q*:	INT := 30000;
	q_nVAG2		AT %Q*:	INT := 30000;
	q_nVAG3		AT %Q*:	INT := 30000;
	q_nVAGF1	AT %Q*:	INT := 30000;
	q_nVAGF2	AT %Q*:	INT := 30000;
	q_nVAGG1	AT %Q*:	INT := 30000;
	q_nVAGG2	AT %Q*:	INT := 30000;
	
	// Used for simulated toggle signal
	pSim:	FB_CRYO_SIM_PRESSURE;
	
	q_nCouplerState	AT %Q*:	INT := 8;
	
	///////////////////////
	// Pressure Ramp Test
	///////////////////////
	SIM_P1:		FB_CRYO_SIM_PRESSURE;
	bStartRamp:	BOOL;
	
	// Actuator test
	actuator:	FB_CRYO_BIN_ACT;
	
	// FB_CRYO_ACTUATOR_CMD test
	Valve1:		FB_CRYO_VALVE_CTRL;		// No override possible
	Valve2:		FB_CRYO_VALVE_CTRL;		// Override possible
	cmdValve2:	FB_CRYO_ACTUATOR_CMD;	// Handling of Valve2 command
	// System commands for Valve1 and Valve2
	bEnable_Valve1:	BOOL;
	bEnable_Valve2:	BOOL;
	
	// FB_CRYO_CMD_OVERRIDE test
	cmdOverrideTest:	FB_CRYO_CMD_OVERRIDE;
	bEnable_OverrideTest:	BOOL;

	//////////////////////////////
	// Testing FB_CRYO_LN2_PRECOOL
	//////////////////////////////
	ln2_ctrl:			FB_CRYO_LN2_PRECOOL;	// LN2 controller
	SIM_ln2:			FB_SIM_LN2_PRECOOL;		// LN2 temperature simulator
	bEnable_ln2_ctrl:	BOOL;					// Flag to activate/deactivate LN2 controller
	
	/////////////////////////////////////////////
	// Testing IO-Link FB_CRYO_SBG232 Flowmeter
	/////////////////////////////////////////////
	
	sbg232:		FB_CRYO_SBG232;
	sbg232_sim:	FB_CRYO_SBG232;
	
	SIM_sbg232:	FB_CRYO_SIM_SBG232;
	
END_VAR

	
Cryo_Ctrl();

SIM_Cryo_Ctrl(in_ptr_Cryo_Ctrl:=ADR(Cryo_Ctrl));


//
// Pressure voting system testing
//
SIM_Pressure_P1(in_nType:=E_CRYO_SENSOR_TYPE_PRESS.PKR_360);


// Measuring point P1 - five sensors
P1_1(in_nType:=E_CRYO_SENSOR_TYPE_PRESS.PKR_360, in_nSampleTime:=100);
P1_2(in_nType:=E_CRYO_SENSOR_TYPE_PRESS.PKR_360, in_nSampleTime:=100);
P1_3(in_nType:=E_CRYO_SENSOR_TYPE_PRESS.PKR_360, in_nSampleTime:=100);
P1_4(in_nType:=E_CRYO_SENSOR_TYPE_PRESS.PKR_360, in_nSampleTime:=100);
P1_5(in_nType:=E_CRYO_SENSOR_TYPE_PRESS.PKR_360, in_nSampleTime:=100);

pressOR_P1(in_bEnable:=bP1_Sim);	// Override of simulation flag
P1(	in_bSimulation	:= pressOR_P1.out_bEnable,
	in_nNumSensor	:= 5, 
	in_nVoteMethod	:= nVoteMethod,
	in_pSensor1		:= ADR(P1_1),
	in_pSensor2		:= ADR(P1_2),
	in_pSensor3		:= ADR(P1_3),
	in_pSensor4		:= ADR(P1_4),
	in_pSensor5		:= ADR(P1_5));

	
//
// Temperature testing
//
T1(in_nRampPeriodSec:=nRampPeriodSec);
tempOR_T2(in_bEnable:=simT2);
T2(in_bSimulation:=tempOR_T2.out_bEnable);


//
// Threshold testing
//
// Simulated sensor value is the combination of two 
// sine wave curves with different period and amplitude.
SIM_thld1(in_lrAmplitude := 95.0, in_nPeriod := nSimPer1);
SIM_thld2(in_lrAmplitude := 20.0, in_nPeriod := nSimPer2);

// Threshold instance
// in_lrValue is the sum of two curves.
thld1(
	in_nMode		:= nThldMode,
	in_aThld		:= aThlds,
	in_aThldDelay	:= aThldDelay,
	in_lrHyst 		:= lrHyst,
	in_lrValue 		:= SIM_thld1.out_lrValue + SIM_thld2.out_lrValue,
	in_lrPar1		:= lrThldRef);


///////////////////
// Lakeshore 336
///////////////////
LS336_TCP(	in_sName			:= 'LS336_TCP',		// Device name
			in_bSimulation		:= FALSE,			// Device simulation
			in_bAutoMonitor		:= TRUE,			// Go to OPERATIONAL, a MUST!
			in_nModel			:= 336,				// Model number
			in_nPeriod			:= 1000,			// Update period [ms]
			in_sCmdSuffix		:= '$0A',			// Command suffix LF
			in_sReplySuffix		:= '$0A',			// Reply suffix LF
			in_sDeviceTcpIpAdr	:= '192.168.0.80', 	// Lakeshore IP address
			in_nDeviceTcpPort	:= 7777);			// Lakeshore port

(*
// Configure Lakeshore for Warmup.
// To be executed only once at the start of the warmup.
LS336_TCP.M_RampEnable(
	in_nPID_A_P			:= 10, 
	in_nPID_A_I			:= 50, 
	in_nPID_A_D			:= 20, 
	in_nHeater_Range	:= 4, 
	in_lrCtrlRamp		:= 1.0, 	// 1.0 deg/min
	in_lrSetpoint_A		:= 293.15);	// 20 deg Celsius
*)			
	
	
///////////////////////////////////////////////////////////////////
// Pumps code
///////////////////////////////////////////////////////////////////
// Handle ELT Cryo Lab Cryostat pressure
cryo_lab_press1(in_nType := E_CRYO_SENSOR_TYPE_PRESS.PKR_250, in_nSampleTime := 100);
cryo_lab_pressure(
	in_bSimulation	:= bSim_cryo_lab_pressure,
	in_nNumSensor	:= 2,	// In reality, there is only one pressure sensor connected
	in_nVoteMethod	:= E_CRYO_VOTE.V_1oo2,
	in_pSensor1		:= ADR(cryo_lab_press1));



// Evacuation system for the PDS IR Imager
evac_pds(in_bEnable	:= bEnable_evac_pds);

// Evacuation system in the ELT Cryo Lab
evac_lab(
	in_bEnable			:= bEnable_evac_lab, 
	in_lrCryoPressure	:= cryo_lab_pressure.stat.lrPressure);


//////////////////////////////
// SUNPOWER Cryotel GT Cooler
//////////////////////////////
cooler(	in_sName		:= 'CryotelGT',
		in_bSimulation	:= TRUE,
		in_bAutoMonitor	:= TRUE,
		in_bEnable		:= bEnable_cooler);

	
	
///////////////
// MICADO
///////////////

pSim();	// Just to have a simulated Toggle signal.

// Simulation of MICADO valves
mic_valves();	

// Simulation of MICADO pumps
mic_pumps(in_RefPVP:=evac_micado.rp, in_RefTMP:=evac_micado.tp);	



// MICADO Cryostat pressures
sensor_VAGF1(in_nType := E_CRYO_SENSOR_TYPE_PRESS.PKR_360,	in_nSampleTime := 100);
sensor_VAGF2(in_nType := E_CRYO_SENSOR_TYPE_PRESS.PKR_360,	in_nSampleTime := 100);
sensor_VAGG1(in_nType := E_CRYO_SENSOR_TYPE_PRESS.PKR_360,	in_nSampleTime := 100);
sensor_VAGG2(in_nType := E_CRYO_SENSOR_TYPE_PRESS.PKR_360,	in_nSampleTime := 100);

VAGF(
	in_bSimulation	:= FALSE,
	in_nNumSensor	:= 2,
	in_nVoteMethod	:= E_CRYO_VOTE.V_1oo2,
	in_pSensor1		:= ADR(sensor_VAGF1),
	in_pSensor2		:= ADR(sensor_VAGF2));

VAGG(
	in_bSimulation	:= FALSE,
	in_nNumSensor	:= 2,
	in_nVoteMethod	:= E_CRYO_VOTE.V_1oo2,
	in_pSensor1		:= ADR(sensor_VAGG1),
	in_pSensor2		:= ADR(sensor_VAGG2));

	
// MICADO evacuation system
cmdPVV1(in_bEnable:=bCmdPVV1,in_bInterlock:=bIntlkPVV1);	// Handling of PVV1 commands

evac_micado(
	in_bEnable		:= bEnable_evac_mic,
	in_RefVAGF		:= VAGF, 
	in_RefVAGG		:= VAGG);
	

///////////////////////
// Pressure Ramp Test
///////////////////////
SIM_P1(	in_nType			:= E_CRYO_SENSOR_TYPE_PRESS.PKR_250, 
		in_lrBitsPerVolt	:= 3276.8, 
		in_lrPress			:= 777.0, 
		in_nPeriod			:= 10000);

// Start ramping from 100 to 0.0001 over 20 sec.
IF bStartRamp	THEN
	bStartRamp	:= FALSE;
	SIM_P1.M_SetValue(100.0);
	SIM_P1.M_RampTo(0.0001,20000);
END_IF
	
// Actuator test
actuator();
	
//
// FB_CRYO_ACTUATOR_CMD test.
//
// Allow only OPEN command for Valve2
cmdValve2.M_SetPermissions(in_bPermitOn := TRUE, in_bPermitOff := FALSE);
// Handling of Valve2 command with active interlock.
cmdValve2(in_bEnable := bEnable_Valve2, in_bInterlock := TRUE);	

Valve1(in_bEnable := bEnable_Valve1);		// Take system command as it is.
Valve2(in_bEnable := cmdValve2.out_bEnable);// Allow user to override system command.

//
// FB_CRYO_CMD_OVERRIDE Test
//
cmdOverrideTest(in_bEnable:=bEnable_OverrideTest);


//////////////////////////////
// Testing FB_CRYO_LN2_PRECOOL
//////////////////////////////
ln2_ctrl(
	in_bEnable		:= bEnable_ln2_ctrl, 
	in_lrTempK		:= SIM_ln2.lrTempK, 
	in_bTempValid	:= TRUE);

SIM_ln2(ln2Ref := ln2_ctrl);


/////////////////////////////////////////////
// Testing IO-Link FB_CRYO_SBG232 Flowmeter
/////////////////////////////////////////////
sbg232();

sbg232_sim(in_sName:='SBG232 SIM');
SIM_sbg232();

END_PROGRAM

// ---- POUs/System/FB_CRYO_CTRL.TcPOU
// Cryogenic Controller Example - ESO IRATEC
FUNCTION_BLOCK FB_CRYO_CTRL
VAR_INPUT
END_VAR
VAR

	///////////////////////////
	// Configuration parameters
	///////////////////////////
	cfg:	T_CRYO_CFG;
	
	/////////////////////
	// Control parameters
	/////////////////////
	ctrl:	T_CRYO_CTRL;

	/////////////////////
	// Status parameters
	/////////////////////
	stat:	T_CRYO_STAT;


	/////////////////////
	// System Logging
	/////////////////////
	syslog:	T_CRYO_LOG;


	/////////////////////
	// Local variables
	/////////////////////



	{attribute 'OPC.UA.DA' := '0'}
	timer:		TON;		// Timer for commands
	
	{attribute 'OPC.UA.DA' := '0'}
	ptrLog:		ARRAY [0..9] OF POINTER TO STRING(80);
	{attribute 'OPC.UA.DA' := '0'}
	nLogPos:	INT := -1;
	
	

//////////////////////////////////////////////
//             Controllers
//////////////////////////////////////////////

//
// LN2 Valve control
//
	{attribute 'OPC.UA.DA' := '1'}
	LN2: 			FB_CRYO_LN2_CTRL;
	
//
// Repressurizing Valve control
//
	{attribute 'OPC.UA.DA' := '1'}
	RepressValve:	FB_CRYO_VALVE_CTRL;
	
	
//
// Evacuation Valve control
//
	EvacSys:	FB_CRYO_EVACUATION_SYSTEM;

//
// Heater control
//
	{attribute 'OPC.UA.DA' := '1'}
	Heater: 		FB_CRYO_HEATER_CTRL;
	
//
// CCC control
//
	{attribute 'OPC.UA.DA' := '1'}
	CCC:			FB_CRYO_CCC_CTRL;

//
// CCC control
//
//	{attribute 'OPC.UA.DA' := '1'}
	Lakeshore:		FB_LAKESHORE_RS;
	
	// Compressor	
	cpa:	FB_CRYO_CPA;

//////////////////////////////////////////////
//             Sensors
//////////////////////////////////////////////
 
//
// VACUUM Sensors
//
	{attribute 'OPC.UA.DA' := '1'}
	Pressure_Cryo:		FB_CRYO_PRESSURE;	
	{attribute 'OPC.UA.DA' := '1'}
	Pressure_Evac:		FB_CRYO_PRESSURE;	
	
 
///////////////////////////////////////////////////////
//                  Temperatures
///////////////////////////////////////////////////////
 
//
// PT100 Temperatures
//
	Temp_Ambient:		FB_CRYO_TEMPERATURE;	// Ambient temperature
	Temp_ColdBench:		FB_CRYO_TEMPERATURE;	// Cold Bench temperature
	Temp_LN2_Exhaust:	FB_CRYO_TEMPERATURE;	// LN2 Exhaust temperature
	Temp_LN2_Inlet:		FB_CRYO_TEMPERATURE;	// LN2 Inlet   temperature
	Temp_Mirror:		FB_CRYO_TEMPERATURE;	// Entrance Mirror temperature
	Temp_WarmUp:		FB_CRYO_TEMPERATURE;	// Reference temperature for WarmUp

//
// Lakeshore temperatures
//
	Temp_DET:			FB_CRYO_TEMPERATURE;	// Lakeshore Channel A
	Temp_HeatShield:	FB_CRYO_TEMPERATURE;	// Heat Shield Lakeshore Channel B
 
//
// IRATEC specific Temperatures
//
	Temp_FW:			FB_CRYO_TEMPERATURE;	// Filter Wheel temperature

	

//
// System triggers
//	
	{attribute 'OPC.UA.DA' := '0'}
	trgPrecool:			R_TRIG;
	{attribute 'OPC.UA.DA' := '0'}
	trgCool:			R_TRIG;
	{attribute 'OPC.UA.DA' := '0'}
	trgWarmup:			R_TRIG;
	{attribute 'OPC.UA.DA' := '0'}
	trgRepress:			R_TRIG;
	{attribute 'OPC.UA.DA' := '0'}
	trgEvacOn:			R_TRIG;
	{attribute 'OPC.UA.DA' := '0'}
	trgEvacOff:			F_TRIG;

//
//	Input signals
//	
	i_bEvacRootPumpOK		AT%I*:	BOOL;
	i_bEvacTurboPumpOK		AT%I*:	BOOL;
	i_bEmergencySTOP		AT%I*:	BOOL;
	i_bManualOverride		AT%I*:	BOOL;
	i_bVacPumpConnected		AT%I*:	BOOL;
	i_bLN2TankConnected		AT%I*:	BOOL;
	i_bRepressLN2Connected	AT%I*:	BOOL;


//
// Dummy values for simulation, etc.
//
	// Dummy OP state for mapping of simulated devices.
	q_nStateDummy	AT%Q*:	UINT := 8;		

	
END_VAR

// Increment cycle counter
stat.nCycleCounter := stat.nCycleCounter + 1;

// Wait until the controller is configured.
IF NOT stat.bConfigured THEN
	M_Configure(); 
	RETURN;
END_IF


//
// Read Temperature and Pressure Sensors
//
M_ReadSensors();


//
// Check for sensor HW errors
//
M_CheckForSensorErrors();



///////////////////
// System Operation
///////////////////

//
// Execute Controllers
//
M_ExecuteControllers();


//
// Capture system commands
//
M_CheckForCommands();


//
// Perform a safety check
//
M_SafetyCheck();


//
// Execute system state machine
//
M_StateMachine();

METHOD M_CheckForCommands
VAR_INPUT
END_VAR
// Capture precooling command
trgPrecool(CLK := ctrl.bEnable_Precool);
IF	trgPrecool.Q AND 
	(stat.nState = E_CRYO_CTRL_STATE.WARM_VACUUM OR stat.nState = E_CRYO_CTRL_STATE.PRE_COOLED) THEN
	ctrl.bExecute	:= TRUE;
	ctrl.nCommand	:= E_CRYO_CTRL_CMD.PRECOOL;
END_IF


// Capture Cool command
trgCool(CLK := ctrl.bEnable_Cool);
IF	trgCool.Q AND stat.nState = E_CRYO_CTRL_STATE.PRE_COOLED THEN
	ctrl.bExecute	:= TRUE;
	ctrl.nCommand	:= E_CRYO_CTRL_CMD.COOL;
END_IF


// Capture Warmup command
trgWarmup(CLK := ctrl.bEnable_Warmup);
IF	trgWarmup.Q AND 
	(stat.nState = E_CRYO_CTRL_STATE.PRE_COOLED OR stat.nState = E_CRYO_CTRL_STATE.COLD) THEN
	ctrl.bExecute	:= TRUE;
	ctrl.nCommand	:= E_CRYO_CTRL_CMD.WARM_UP;
END_IF


// Capture Repressure command
trgRepress(CLK := ctrl.bEnable_RepressCtrl);
IF	trgRepress.Q AND 
	(stat.nState = E_CRYO_CTRL_STATE.WARM_VACUUM) THEN
	ctrl.bExecute	:= TRUE;
	ctrl.nCommand	:= E_CRYO_CTRL_CMD.REPRESSURIZE;
END_IF


// Capture Evacuation ON/OFF trigger
trgEvacOn(CLK := ctrl.bEnable_Evac);
trgEvacOff(CLK := ctrl.bEnable_Evac);
IF	trgEvacOn.Q AND NOT ctrl.bEnable_RepressSys THEN
	ctrl.bEnable_Evac	:= TRUE;
	M_SysLog('Evacuation started.');
ELSIF trgEvacOff.Q THEN
	ctrl.bEnable_Evac	:= FALSE;
	M_SysLog('Evacuation stopped.');
END_IF
END_METHOD

METHOD M_CheckForSensorErrors
VAR_INPUT
END_VAR
////////////////////////////////////////////////
// Check for errors by testing the 'Valid' flag.
////////////////////////////////////////////////
IF		NOT Pressure_Cryo.stat.bValid	THEN
	stat.bError	:= TRUE;
	stat.sState	:= 'Cryo Vacuum gauge problem';
	stat.nState	:= E_CRYO_CTRL_STATE.ERROR;
ELSIF	NOT Temp_Mirror.stat.bValid	THEN
	stat.bError	:= TRUE;
	stat.sState	:= 'Mirror Temperature sensor problem';
	stat.nState	:= E_CRYO_CTRL_STATE.ERROR;
ELSE
	stat.bError	:= FALSE;
	stat.sState	:= '';
END_IF


///////////////////////
// Check for Interlocks
///////////////////////

//
// Evacuation and Repressurization are mutually exclusive.
//
IF EvacSys.in_bEnable THEN
	ctrl.bEnable_RepressSys	:= FALSE;
ELSIF RepressValve.in_bEnable THEN
	ctrl.bEnable_Evac	:= FALSE;
END_IF

//
// Disable control in failure state
//
IF stat.bError THEN
	ctrl.bEnable_Precool	:= FALSE;
	ctrl.bEnable_Cool 		:= FALSE;
	ctrl.bEnable_Warmup		:= FALSE;
END_IF
END_METHOD

METHOD M_CheckLakeshoreCommand
VAR_INPUT
END_VAR
(* TODO

IF ctrl.bLS_UpdateSETP THEN
	// Reset trigger flag
	ctrl.bLS_UpdateSETP	:= FALSE;
	
	// Safety
	IF ctrl.lrLS_RAMP > 1.0 THEN
		ctrl.lrLS_RAMP	:= 1.0;
	ELSIF ctrl.lrLS_RAMP < 0.0 THEN
		ctrl.lrLS_RAMP	:= 0.0;
	END_IF
	
	// Set the mode
	IF ctrl.nLS_Mode <> E_CRYO_LAKESHORE_MODE.MONITORING THEN
		Lakeshore.M_SetMode(ctrl.nLS_Mode);
	ELSE
		RETURN;	// Nothing to do
	END_IF
ELSE
	RETURN;	// Nothing to do
END_IF




CASE ctrl.nLS_Mode OF
	E_CRYO_LAKESHORE_MODE.MONITORING,
	E_CRYO_LAKESHORE_MODE.COOLING,
	E_CRYO_LAKESHORE_MODE.WARMUP,
	E_CRYO_LAKESHORE_MODE.COOLING_UPDATE,
	E_CRYO_LAKESHORE_MODE.WARMUP_UPDATE:
		Lakeshore.M_SetMode(E_CRYO_LAKESHORE_MODE.MONITORING);	// No action
		
	E_CRYO_LAKESHORE_MODE.SINGLE_SETUP:
		IF stat.nState = E_CRYO_CTRL_STATE.COLD THEN
			Lakeshore.M_SetParams(
				in_nPID_A_P			:= cfg.LS_W_PID_A_P, 
				in_nPID_A_I			:= cfg.LS_W_PID_A_I, 
				in_nPID_A_D			:= cfg.LS_W_PID_A_D, 
				in_nHeater_Range	:= cfg.LS_W_Heater_Range, 
				in_lrCtrlRamp		:= ctrl.lrLS_RAMP, 
				in_lrSetpoint_A		:= ctrl.lrLS_SETP);
		END_IF
	ELSE
		Lakeshore.M_SetMode(E_CRYO_LAKESHORE_MODE.MONITORING);	// No action
END_CASE
*)
END_METHOD

// Method to check status of the cryostat vacuum.
// TODO: The limits might depend on the temperature.
METHOD M_CheckVacuum
VAR_INPUT
END_VAR
IF Pressure_Cryo.stat.bValid  THEN
	IF Pressure_Cryo.stat.lrPressure < cfg.lrPress_GoodVac THEN
		stat.bInVacuum	:= TRUE;
		stat.bGoodVacuum:= TRUE;
	ELSIF Pressure_Cryo.stat.lrPressure < cfg.lrPress_InVac THEN
		stat.bInVacuum	:= TRUE;
		stat.bGoodVacuum:= FALSE;
	ELSE
		stat.bInVacuum	:= FALSE;
		stat.bGoodVacuum:= FALSE;
	END_IF 
ELSE
	stat.bInVacuum	:= FALSE;
	stat.bGoodVacuum:= FALSE;
END_IF
END_METHOD

METHOD M_Configure
VAR_INPUT
END_VAR
IF stat.bConfigured THEN
	RETURN;
ELSIF stat.nCycleCounter = 100 THEN
	// Set pointers to system logs.
	ptrLog[0] := ADR(syslog.s0);
	ptrLog[1] := ADR(syslog.s1);
	ptrLog[2] := ADR(syslog.s2);
	ptrLog[3] := ADR(syslog.s3);
	ptrLog[4] := ADR(syslog.s4);
	ptrLog[5] := ADR(syslog.s5);
	ptrLog[6] := ADR(syslog.s6);
	ptrLog[7] := ADR(syslog.s7);
	ptrLog[8] := ADR(syslog.s8);
	ptrLog[9] := ADR(syslog.s9);
ELSIF stat.nCycleCounter > 200 THEN
	stat.bConfigured	:= TRUE;
ELSE
	RETURN;
END_IF
END_METHOD

METHOD M_ExecuteControllers
VAR
END_VAR
//
// Controllers, i.e. LN2 cooler, Heater, ...
//

// Activate Lakeshore SETP command, if any (see ctrl.xxLS_...)
M_CheckLakeshoreCommand();

// Execute Lakeshore 340 controller
Lakeshore(
	in_bSimulation	:= TRUE,
	in_sName		:= 'LS340',
	in_nModel		:= 340, 
	in_bAutoMonitor	:= TRUE, 
	in_nPeriod 		:= 2000,
	in_sCmdSuffix	:= '$0D$0A',
	in_sReplySuffix	:= '$0D$0A');


LN2(
	in_bEnable			:= ctrl.bEnable_Precool, 
	in_nFeedback		:= E_CRYO_BIN_ACT_FEEDBACK.ON_ONLY, 
	in_lrTempK			:= Temp_LN2_Exhaust.stat.lrTempK, 
	in_bValid			:= Temp_LN2_Exhaust.stat.bValid, 
	in_lrTempValveOpen	:= cfg.lrTemp_LN2ValveOpen, 
	in_lrTempValveClose	:= cfg.lrTemp_LN2ValveClose);
	
RepressValve(in_bEnable	:= ctrl.bEnable_RepressCtrl);
	
EvacSys(
	in_bEnable			:= ctrl.bEnable_Evac,
	in_Pressure_Cryo	:= Pressure_Cryo.stat,
	in_Pressure_Evac	:= Pressure_Evac.stat,
	in_Temp_Cryo		:= Temp_Mirror.stat,
	in_bRepressValveOpen:= RepressValve.stat.bActON, 
	in_bRepressValveOK	:= NOT RepressValve.stat.bError);

	
// Heater compares DET temperature against the lowest temperature in the system. 
// Lowest temperature is calculated in M_ReadSensors() by 
// calling M_GetLowestTemperature().
Heater(
	in_bEnable		:= (ctrl.bEnable_Heater AND NOT i_bEmergencySTOP), 
	in_nFeedback	:= E_CRYO_BIN_ACT_FEEDBACK.ON_ONLY, 
	in_lrTemp1		:= stat.lrHighestTempK, 
	in_lrTemp2		:= Temp_DET.stat.lrTempK, 
	in_bValidTemp1	:= stat.bHighestTempValid,
	in_bValidTemp2	:= Temp_DET.stat.bValid,
	in_lrDelta_Low	:= cfg.lrTemp_DeltaDet_Bench_Low, 
	in_lrDelta_High	:= cfg.lrTemp_DeltaDet_Bench_High);

	
CCC(in_bEnable	:= ctrl.bEnable_CCC);


cpa(in_bSimulation				:= FALSE,
	in_sName					:= 'PT810-01',
	in_sSN_Compressor			:= 'CPA289C-W2EHCE-180201A',
	in_sSN_PulseTube			:= 'CH40810-180208A',
	in_nYear_Compressor			:= 2018,
	in_nYear_PulseTube			:= 2020,
	in_lrNextService_Compressor	:= 20000.0,
	in_lrNextService_PulseTube	:= 35000.0,
	in_nSlaveID					:= 16,
	in_nPeriod					:= 1000);
END_METHOD

METHOD M_GetHighestTemperature
VAR_INPUT
END_VAR
VAR
	lrTempK:	LREAL	:= 0.0;	// The lowest possible temperature
	bValid:		BOOL	:= FALSE;
END_VAR
//
// Get the warmest temperature among Mirror, Bench, FilterWheel and WarmUp
//

// If there is at least one Valid reading, the result is valid.
IF	Temp_Mirror.stat.bValid 	OR 
	Temp_ColdBench.stat.bValid	OR 
	Temp_FW.stat.bValid			OR 
	Temp_WarmUp.stat.bValid			THEN
	bValid	:= TRUE;
END_IF


// Get the highest temperature from Valid temperatures.
// Take Mirror temperature first, if Valid.
// If not Valid, try with WarmUp sensor.
// If that doesn't work, take the Filter Wheel temperature.
IF Temp_Mirror.stat.bValid THEN
	IF Temp_Mirror.stat.lrTempK > lrTempK THEN
		lrTempK	:= Temp_Mirror.stat.lrTempK;
	END_IF
ELSIF Temp_WarmUp.stat.bValid THEN
	IF Temp_WarmUp.stat.lrTempK > lrTempK THEN
		lrTempK	:= Temp_Mirror.stat.lrTempK;
	END_IF
ELSIF Temp_FW.stat.bValid THEN
	IF Temp_FW.stat.lrTempK > lrTempK THEN
		lrTempK	:= Temp_Mirror.stat.lrTempK;
	END_IF
END_IF


// Update status
stat.lrHighestTempK		:= lrTempK;
stat.bHighestTempValid	:= bValid;
END_METHOD

METHOD M_GetLowestTemperature
VAR_INPUT
END_VAR
VAR
	lrTempK:	LREAL	:= 293.15;	// Room temperature 20 C
	bValid:		BOOL	:= FALSE;
END_VAR
//
// Get the coldest temperature among Mirror, Bench, FilterWheel and WarmUp
//

// If there is at least one Valid reading, the result is valid.
IF	Temp_Mirror.stat.bValid 	OR 
	Temp_ColdBench.stat.bValid	OR 
	Temp_FW.stat.bValid			OR 
	Temp_WarmUp.stat.bValid			THEN
	bValid	:= TRUE;
END_IF


// Get the lowest temperature from Valid temperatures.
IF Temp_Mirror.stat.bValid AND Temp_Mirror.stat.lrTempK < lrTempK THEN
	lrTempK	:= Temp_Mirror.stat.lrTempK;
END_IF

IF Temp_ColdBench.stat.bValid AND Temp_ColdBench.stat.lrTempK < lrTempK THEN
	lrTempK	:= Temp_ColdBench.stat.lrTempK;
END_IF

IF Temp_FW.stat.bValid AND Temp_FW.stat.lrTempK < lrTempK THEN
	lrTempK	:= Temp_FW.stat.lrTempK;
END_IF

IF Temp_WarmUp.stat.bValid AND Temp_WarmUp.stat.lrTempK < lrTempK THEN
	lrTempK	:= Temp_WarmUp.stat.lrTempK;
END_IF

// Update status
stat.lrLowestTempK		:= lrTempK;
stat.bLowestTempValid	:= bValid;

// Get Temperature difference (DET -Lowest temperature) [K]
IF stat.bLowestTempValid  AND  Temp_DET.stat.bValid  THEN
	stat.bDiffTempValid	:= TRUE;
	stat.lrDiffTempK	:= Temp_DET.stat.lrTempK - stat.lrLowestTempK;
ELSE
	stat.bDiffTempValid	:= FALSE;
	stat.lrDiffTempK	:= -100;
END_IF
END_METHOD

METHOD M_GetState
VAR_INPUT
END_VAR
// Determine the initial state based on the command and actuator state.
IF NOT stat.bCtrlOK	THEN
	stat.nState	:= E_CRYO_CTRL_STATE.ERROR;
ELSIF	Temp_Mirror.stat.lrTempK >= cfg.lrTemp_Precooled  AND  NOT stat.bInVacuum	THEN
	stat.nState	:= E_CRYO_CTRL_STATE.WARM_PRESS;
ELSIF	Temp_Mirror.stat.lrTempK >= cfg.lrTemp_Precooled  AND  stat.bInVacuum  THEN
	stat.nState	:= E_CRYO_CTRL_STATE.WARM_VACUUM;
ELSIF	Temp_Mirror.stat.lrTempK < cfg.lrTemp_Cold 	AND  stat.bInVacuum  THEN
	stat.nState	:= E_CRYO_CTRL_STATE.COLD;
ELSIF	Temp_Mirror.stat.lrTempK < cfg.lrTemp_Precooled  AND  stat.bInVacuum  THEN
	stat.nState	:= E_CRYO_CTRL_STATE.PRE_COOLED;
END_IF
M_SetStatus(stat.nState);
END_METHOD

METHOD M_ReadSensors
VAR_INPUT
END_VAR
//
// Read system temperatures, i.e. LN2, Bench and Detector temperatures
//
Temp_Ambient		(in_lrScale_1:=0.1);
Temp_ColdBench 		(in_lrScale_1:=0.1, in_bIgnoreUnderrange_1 := ctrl.bIgnoreUnderrange_ColdBench);
Temp_LN2_Exhaust	(in_lrScale_1:=0.1);
Temp_LN2_Inlet		(in_lrScale_1:=0.1);
Temp_Mirror			(in_lrScale_1:=0.1);
Temp_WarmUp			(in_lrScale_1:=0.1);

Temp_FW				(in_lrScale_1:=0.1);	// IRATEC specific

//
// Lakeshore temperature
//
// Important note:
// In normal operation, call to Temp_DET() will result in a reading that is
// not valid since the underlying temperature sensors should not be 
// mapped to temperature signals.
// However, call to Temp_DET.M_GetTemperatureFromLakeshore() will copy 
// the Lakeshore reading to it and update the Valid flag.
//
// DET temperature is Lakeshore Channel A

(* TODO
Temp_DET(in_lrScale_1:=0.1);	
Temp_DET.M_GetTemperatureFromLakeshore(
	bValid	:= (Lakeshore.stat.nErrorCode=0),
	lrTempK	:=  Lakeshore.stat.lrKRDG_A,
	lrTempC	:=  Lakeshore.stat.lrCRDG_A);

// HeatShield temperature is Lakeshore Channel B
Temp_HeatShield(in_lrScale_1:=0.1);
Temp_HeatShield.M_GetTemperatureFromLakeshore(
	bValid	:= (Lakeshore.stat.nErrorCode=0),
	lrTempK	:=  Lakeshore.stat.lrKRDG_B,
	lrTempC	:=  Lakeshore.stat.lrCRDG_B);

*)

// Both pressure sensors are of PKR250/251 type
Pressure_Cryo(	in_lrLimitInVac		:= cfg.lrPress_InVac, 
				in_lrLimitGoodVac	:= cfg.lrPress_GoodVac);
Pressure_Evac(	in_lrLimitInVac		:= cfg.lrPress_InVac, 
				in_lrLimitGoodVac	:= cfg.lrPress_GoodVac);	

//
// Get the lowest temperature in the cryostat
//	
M_GetLowestTemperature();

//
// Get the highest temperature in the cryostat
//	
M_GetHighestTemperature();
	

//
// Check Vacuum in the system
//	
M_CheckVacuum();
END_METHOD

METHOD M_SafetyCheck
VAR_INPUT
END_VAR
//
// Repressurization safety
//
IF	NOT ctrl.bEnable_Evac AND
	(stat.nState = E_CRYO_CTRL_STATE.WARM_PRESS 		OR 
	 stat.nState = E_CRYO_CTRL_STATE.REPRESSURIZING 	OR 
	 stat.nState = E_CRYO_CTRL_STATE.WARM_VACUUM) 		THEN
	ctrl.bSafe_Repress	:= TRUE;
ELSE
	ctrl.bSafe_Repress	:= FALSE;
	ctrl.bEnable_RepressSys:= FALSE;
END_IF
END_METHOD

METHOD M_SetStatus
VAR_INPUT
	nState:	E_CRYO_CTRL_STATE;
END_VAR

CASE nState OF
	
	E_CRYO_CTRL_STATE.NONE:
	stat.bDone	:= TRUE;
	stat.bBusy	:= FALSE;
	stat.bError	:= FALSE;
	stat.bActive:= FALSE;
	stat.sState	:= 'OFF';
	
	E_CRYO_CTRL_STATE.WARM_PRESS:
	stat.bDone	:= TRUE;
	stat.bBusy	:= FALSE;
	stat.bError	:= FALSE;
	stat.bActive:= TRUE;
	stat.sState	:= 'WARM  -  PRESSURIZED';
	
	E_CRYO_CTRL_STATE.WARM_VACUUM:
	stat.bDone	:= TRUE;
	stat.bBusy	:= FALSE;
	stat.bError	:= FALSE;
	stat.bActive:= TRUE;
	stat.sState	:= 'WARM  -  VACUUM';
	
	E_CRYO_CTRL_STATE.PRE_COOLING:
	stat.bDone	:= FALSE;
	stat.bBusy	:= TRUE;
	stat.bError	:= FALSE;
	stat.bActive:= TRUE;
	stat.sState	:= 'PRE-COOLING...';
	
	E_CRYO_CTRL_STATE.PRE_COOLED:
	stat.bDone	:= TRUE;
	stat.bBusy	:= FALSE;
	stat.bError	:= FALSE;
	stat.bActive:= TRUE;
	stat.sState	:= 'PRE-COOLED';

	E_CRYO_CTRL_STATE.COOLING_DOWN:
	stat.bDone	:= FALSE;
	stat.bBusy	:= TRUE;
	stat.bError	:= FALSE;
	stat.bActive:= TRUE;
	stat.sState	:= 'COOLING DOWN...';

	E_CRYO_CTRL_STATE.COLD:
	stat.bDone	:= TRUE;
	stat.bBusy	:= FALSE;
	stat.bError	:= FALSE;
	stat.bActive:= TRUE;
	stat.sState	:= 'COLD';

	E_CRYO_CTRL_STATE.WARMING_UP:
	stat.bDone	:= FALSE;
	stat.bBusy	:= TRUE;
	stat.bError	:= FALSE;
	stat.bActive	:= TRUE;
	IF Temp_Mirror.stat.lrTempK >= cfg.lrTemp_Warm	THEN
		stat.sState	:= 'WARM';
	ELSIF	Temp_Mirror.stat.lrTempK < cfg.lrTemp_Warm AND
			Temp_Mirror.stat.lrTempK >= cfg.lrTemp_Precooled	THEN
		stat.sState	:= 'WARMING UP... PRE-COOLED';
	ELSE
		stat.sState	:= 'WARMING UP... COLD';
	END_IF

	E_CRYO_CTRL_STATE.REPRESSURIZING:
	stat.bDone	:= FALSE;
	stat.bBusy	:= TRUE;
	stat.bError	:= FALSE;
	stat.bActive:= TRUE;
	stat.sState	:= 'RE-PRESSURIZING...';
	
	E_CRYO_CTRL_STATE.ERROR:
	stat.bDone	:= TRUE;
	stat.bBusy	:= FALSE;
	stat.bError	:= TRUE;
	stat.bActive:= FALSE;
	stat.sState	:= 'ERROR';

END_CASE
END_METHOD

METHOD M_StateMachine
VAR_INPUT
END_VAR
////////////////
// State Machine
////////////////
CASE stat.nState OF
	/////////////////////////////////
	E_CRYO_CTRL_STATE.NONE:
	/////////////////////////////////
	//
	// This is the state on power-up.
	// Determine the initial state based on the command and actuator state.
	M_GetState();	
	RETURN;
	

	/////////////////////////////////
	E_CRYO_CTRL_STATE.WARM_PRESS:
	/////////////////////////////////
	//
	ctrl.bSafe_Precool	:= FALSE;
	ctrl.bSafe_Cooling	:= FALSE;
	ctrl.bSafe_Warmup	:= FALSE;

	ctrl.bEnable_RepressCtrl:= FALSE;
	ctrl.bEnable_Heater		:= FALSE;

	IF	ctrl.bExecute	THEN
		ctrl.bExecute		:= FALSE;
		stat.nLastCommand	:= ctrl.nCommand;
		ctrl.nCommand		:= E_CRYO_CTRL_CMD.NONE;
	ELSIF Pressure_Cryo.stat.lrPressure < cfg.lrPress_InVac THEN
		// Evacuation is not part of the State Machine.
		// Once the air has been evacuated, we switch to WARM_VACUUM.
		stat.nState := E_CRYO_CTRL_STATE.WARM_VACUUM;
	END_IF
	M_SetStatus(stat.nState);	
	RETURN;
	
	
	//////////////////////////////////////////
	E_CRYO_CTRL_STATE.WARM_VACUUM:
	//////////////////////////////////////////
	//
	ctrl.bSafe_Precool	:= NOT ctrl.bEnable_RepressSys;
	ctrl.bSafe_Cooling	:= FALSE;
	ctrl.bSafe_Warmup	:= FALSE;
	
	// In this state CCC should be OFF
	ctrl.bEnable_CCC	:= FALSE;
	ctrl.bEnable_Heater	:= FALSE;

	IF	ctrl.bExecute	THEN
		ctrl.bExecute		:= FALSE;
		stat.nLastCommand	:= ctrl.nCommand;
		ctrl.nCommand		:= E_CRYO_CTRL_CMD.NONE;
		IF stat.nLastCommand = E_CRYO_CTRL_CMD.PRECOOL	THEN
			IF CCC.stat.bActive THEN
				ctrl.bEnable_Precool	:= FALSE;
				M_SysLog('Cannot start pre-cooling. CCC still active!');
				RETURN;
			ELSIF CCC.stat.bError THEN
				ctrl.bEnable_Precool	:= FALSE;
				M_SysLog('Cannot start pre-cooling. CCC in Error state!');
				RETURN;
			END_IF
			
			// Configure Lakeshore for Cooling
			Lakeshore.M_RampEnable(
				in_nPID_A_P			:= cfg.LS_C_PID_A_P, 
				in_nPID_A_I			:= cfg.LS_C_PID_A_I, 
				in_nPID_A_D			:= cfg.LS_C_PID_A_D, 
				in_nHeater_Range	:= cfg.LS_C_Heater_Range, 
				in_lrCtrlRamp		:= cfg.LS_C_CTRL_RAMP, 
				in_lrSetpoint_A		:= cfg.LS_C_SETPOINT_A);
			
			M_SysLog('Pre-cooling started.');
			stat.nState	:= E_CRYO_CTRL_STATE.PRE_COOLING;
		ELSIF stat.nLastCommand = E_CRYO_CTRL_CMD.REPRESSURIZE	THEN
			// Disable Evacuation Valve control
			ctrl.bEnable_Evac	:= FALSE;
			ctrl.bEnable_RepressCtrl := TRUE;
			
			// Configure Lakeshore just to monitor. Disable control.
			Lakeshore.M_RampDisable();

			M_SysLog('Re-pressurization started.');
			stat.nState	:= E_CRYO_CTRL_STATE.REPRESSURIZING;
		END_IF
	END_IF
	M_SetStatus(stat.nState);	
	RETURN;
	

	/////////////////////////////////
	E_CRYO_CTRL_STATE.PRE_COOLING:
	/////////////////////////////////
	//
	ctrl.bSafe_Precool	:= TRUE;
	ctrl.bSafe_Cooling	:= FALSE;
	ctrl.bSafe_Warmup	:= FALSE;

	ctrl.bEnable_CCC	:= FALSE;

	ctrl.bEnable_RepressCtrl:= FALSE;

	IF Temp_Mirror.stat.lrTempK < cfg.lrTemp_Precooled	THEN
		M_SysLog('Pre-cooling complete. State is Pre-cooled.');
		stat.nState	:= E_CRYO_CTRL_STATE.PRE_COOLED;
	ELSIF NOT ctrl.bEnable_Precool THEN
		// Pre-cooling has been interrupted.
		// Go back to WARM_VACUUM state.
		M_SysLog('Pre-cooling interrupted. State is Warm-Vacuum.');
		stat.nState := E_CRYO_CTRL_STATE.WARM_VACUUM;
	END_IF
	M_SetStatus(stat.nState);	
	RETURN;
	
	
	///////////////////////////////////////////
	E_CRYO_CTRL_STATE.PRE_COOLED:
	///////////////////////////////////////////
	//
	ctrl.bSafe_Precool	:= TRUE;
	ctrl.bSafe_Cooling	:= NOT ctrl.bEnable_Precool;
	ctrl.bSafe_Warmup	:= NOT ctrl.bEnable_Precool;
	ctrl.bEnable_CCC	:= FALSE;

	ctrl.bEnable_RepressCtrl:= FALSE;

	//
	// Only COOL and WARM_UP commands are allowed in state PRE_COOLED.
	// Other commands are ignored.
	//
	IF	ctrl.bExecute	THEN
		ctrl.bExecute		:= FALSE;
		stat.nLastCommand	:= ctrl.nCommand;
		ctrl.nCommand		:= E_CRYO_CTRL_CMD.NONE;
		IF stat.nLastCommand = E_CRYO_CTRL_CMD.COOL	THEN
			IF LN2.stat.bActive THEN
				M_SysLog('Cannot start cooling. LN2 still active!');
				RETURN;
			ELSIF LN2.stat.bError THEN
				M_SysLog('Cannot start cooling. LN2 in Error state!');
				RETURN;
			END_IF

			// Configure Lakeshore for cooling
			Lakeshore.M_RampEnable(
				in_nPID_A_P			:= cfg.LS_C_PID_A_P, 
				in_nPID_A_I			:= cfg.LS_C_PID_A_I, 
				in_nPID_A_D			:= cfg.LS_C_PID_A_D, 
				in_nHeater_Range	:= cfg.LS_C_Heater_Range, 
				in_lrCtrlRamp		:= cfg.LS_C_CTRL_RAMP, 
				in_lrSetpoint_A		:= cfg.LS_C_SETPOINT_A);
			
			M_SysLog('Cool-down started.');
			stat.nState	:= E_CRYO_CTRL_STATE.COOLING_DOWN;
		ELSIF stat.nLastCommand = E_CRYO_CTRL_CMD.WARM_UP	THEN
			// Eable Evacuation Valve control here.
			// This way the user will be able to turn it on/off
			// during the warmup phase.
			ctrl.bEnable_Evac	:= TRUE;

			// Configure Lakeshore for Warmup
			Lakeshore.M_RampEnable(
				in_nPID_A_P			:= cfg.LS_W_PID_A_P, 
				in_nPID_A_I			:= cfg.LS_W_PID_A_I, 
				in_nPID_A_D			:= cfg.LS_W_PID_A_D, 
				in_nHeater_Range	:= cfg.LS_W_Heater_Range, 
				in_lrCtrlRamp		:= cfg.LS_W_CTRL_RAMP, 
				in_lrSetpoint_A		:= cfg.LS_W_SETPOINT_A);
			
			M_SysLog('Warm-up started.');
			stat.nState	:= E_CRYO_CTRL_STATE.WARMING_UP;
		END_IF
	END_IF
	M_SetStatus(stat.nState);	
	RETURN;
	
	/////////////////////////////////
	E_CRYO_CTRL_STATE.COOLING_DOWN:
	/////////////////////////////////
	//
	ctrl.bSafe_Precool	:= FALSE;
	ctrl.bSafe_Cooling	:= TRUE;
	ctrl.bSafe_Warmup	:= FALSE;
	ctrl.bEnable_CCC	:= TRUE;

	ctrl.bEnable_RepressCtrl:= FALSE;
	
	IF Temp_Mirror.stat.lrTempK < cfg.lrTemp_Cold	THEN
		M_SysLog('Cool-down complete. State is Cold.');
		// Enable Evacuation Valve control
		ctrl.bEnable_Evac	:= TRUE;
		stat.nState	:= E_CRYO_CTRL_STATE.COLD;
	ELSIF NOT ctrl.bEnable_Cool THEN
		// Cooling has been interrupted.
		// Go back to PRE_COOLED state.
		M_SysLog('Cooling interrupted. State is Pre-cooled.');
		stat.nState := E_CRYO_CTRL_STATE.PRE_COOLED;
	END_IF
	M_SetStatus(stat.nState);	
	RETURN;
	
	
	///////////////////////////////////////////
	E_CRYO_CTRL_STATE.COLD:
	///////////////////////////////////////////
	//
	ctrl.bSafe_Precool	:= FALSE;
	ctrl.bSafe_Cooling	:= TRUE;
	ctrl.bSafe_Warmup	:= NOT ctrl.bEnable_Cool;

	ctrl.bEnable_CCC		:= TRUE;
	ctrl.bEnable_RepressCtrl:= FALSE;

	//
	// Only WARM_UP command is allowed in state COLD.
	// Other commands are ignored.
	//
	IF	ctrl.bExecute	THEN
		ctrl.bExecute		:= FALSE;
		stat.nLastCommand	:= ctrl.nCommand;
		ctrl.nCommand		:= E_CRYO_CTRL_CMD.NONE;
		IF stat.nLastCommand = E_CRYO_CTRL_CMD.WARM_UP	THEN
			// Turbo OK
			// CCC OFF - by Hand (button)
			// LN2 OFF
			
			// Eable Evacuation Valve control here.
			// This way the user will be able to turn it on/off
			// during the warmup phase.
			ctrl.bEnable_Evac	:= TRUE;

			// Configure Lakeshore for Warmup
			Lakeshore.M_RampEnable(
				in_nPID_A_P			:= cfg.LS_W_PID_A_P, 
				in_nPID_A_I			:= cfg.LS_W_PID_A_I, 
				in_nPID_A_D			:= cfg.LS_W_PID_A_D, 
				in_nHeater_Range	:= cfg.LS_W_Heater_Range, 
				in_lrCtrlRamp		:= cfg.LS_W_CTRL_RAMP, 
				in_lrSetpoint_A		:= cfg.LS_W_SETPOINT_A);
			
			M_SysLog('Warm-up started.');
			stat.nState	:= E_CRYO_CTRL_STATE.WARMING_UP;
		END_IF
	END_IF
	M_SetStatus(stat.nState);	
	RETURN;
	
	/////////////////////////////////
	E_CRYO_CTRL_STATE.WARMING_UP:
	/////////////////////////////////
	//
	ctrl.bSafe_Precool	:= FALSE;
	ctrl.bSafe_Cooling	:= FALSE;

	ctrl.bEnable_Heater := TRUE;

	// In this state CCC should be OFF
	ctrl.bEnable_CCC	:= FALSE;
	
	// Switch LN2 OFF
	ctrl.bEnable_Precool	:= FALSE;
	
	// Block re-pressurisation subsystem
	ctrl.bEnable_RepressCtrl:= FALSE;

	// TODO: ???
	// Evac.stat.bActON must be all the time. 
	// If not, error AND 
	// ctrl.bEnable_Heater := false; AND
	// Re-configure Lakeshore for IDLE (no warming)

	IF Temp_Mirror.stat.lrTempK > cfg.lrTemp_Warm	THEN
		// Cryo temperature is higher than the Warm threshold.
		// The cryo is in WARM_VACUUM state.
		ctrl.bEnable_Warmup	:= FALSE;
		M_SysLog('Warm-up complete. State is Warm-Vacuum.');
		stat.nState	:= E_CRYO_CTRL_STATE.WARM_VACUUM;
	ELSIF NOT ctrl.bEnable_Warmup THEN
		// Warming up has been interrupted.
		// Based on the Bench temperature determine whether
		// the Cryo is in PRE_COOLED or COLD state.
		IF	Temp_Mirror.stat.lrTempK <  cfg.lrTemp_Warm AND
			Temp_Mirror.stat.lrTempK >= cfg.lrTemp_Precooled	THEN
			// Go back to PRE_COOLED state.
			M_SysLog('Warming up interrupted. State is Pre-cooled.');
			stat.nState := E_CRYO_CTRL_STATE.PRE_COOLED;
		ELSE
			// Go back to COLD state.
			M_SysLog('Warming up interrupted. State is Cold.');
			stat.nState := E_CRYO_CTRL_STATE.COLD;
		END_IF
	END_IF
	M_SetStatus(stat.nState);	
	RETURN;
	
	
	/////////////////////////////////
	E_CRYO_CTRL_STATE.REPRESSURIZING:
	/////////////////////////////////
	//
	ctrl.bSafe_Precool	:= FALSE;
	ctrl.bSafe_Cooling	:= FALSE;
	ctrl.bSafe_Warmup	:= FALSE;

	ctrl.bEnable_CCC	:= FALSE;

